// TIA Portal project "LF_project" (V16)

(* hardware
DEVICE "S7-1200 station_1"  S7-1200 Station
   slot 0: "Rack_0"  S7-1200 Rack  Rack  V1.0
   slot 1: "PLC_1"  CPU 1214C DC/DC/DC  6ES7 214-1AG40-0XB0  V4.2
   slot 2: "DI 16/DQ 16x24VDC_1"  6ES7 223-1BL32-0XB0  V2.0
   slot 3: "DI 16/DQ 16x24VDC_2"  6ES7 223-1BL32-0XB0  V2.0
   slot 4: "DI 16/DQ 16x24VDC_3"  6ES7 223-1BL32-0XB0  V2.0
   slot 5: "DI 16/DQ 16x24VDC_4"  6ES7 223-1BL32-0XB0  V2.0
   slot 6: "DI 16/DQ 16x24VDC_5"  6ES7 223-1BL32-0XB0  V2.0
   slot 7: "DI 16/DQ 16x24VDC_6"  6ES7 223-1BL32-0XB0  V2.0
*)

// ===== PLC "PLC_1"  CPU 1214C DC/DC/DC =====

VAR_GLOBAL   // PLC tag table "Default tag table"
   "System_Byte" AT %MB1 : Byte;
   "FirstScan" AT %M1.0 : Bool;
   "DiagStatusUpdate" AT %M1.1 : Bool;
   "AlwaysTRUE" AT %M1.2 : Bool;
   "AlwaysFALSE" AT %M1.3 : Bool;
END_VAR

VAR_GLOBAL   // PLC tag table "Input tags_1"
   "IN_1-0.0" AT %I0.0 : Bool;
   "IN_1-0.1" AT %I0.1 : Bool;
   "IN_1-0.2" AT %I0.2 : Bool;
   "IN_1-0.3" AT %I0.3 : Bool;
   "IN_1-0.4" AT %I0.4 : Bool;
   "IN_1-0.5" AT %I0.5 : Bool;
   "IN_1-0.6" AT %I0.6 : Bool;
   "IN_1-0.7" AT %I0.7 : Bool;
   "IN_1-1.0" AT %I1.0 : Bool;
   "IN_1-1.1" AT %I1.1 : Bool;
   "IN_1-1.2" AT %I1.2 : Bool;
   "IN_1-1.3" AT %I1.3 : Bool;
   "IN_1-1.4" AT %I1.4 : Bool;
   "IN_1-1.5" AT %I1.5 : Bool;
END_VAR

VAR_GLOBAL   // PLC tag table "Output tags_1"
   "OUT_1-0.0" AT %Q0.0 : Bool;
   "OUT_1-0.1" AT %Q0.1 : Bool;
   "OUT_1-0.2" AT %Q0.2 : Bool;
   "OUT_1-0.3" AT %Q0.3 : Bool;
   "OUT_1-0.4" AT %Q0.4 : Bool;
   "OUT_1-0.5" AT %Q0.5 : Bool;
   "OUT_1-0.6" AT %Q0.6 : Bool;
   "OUT_1-0.7" AT %Q0.7 : Bool;
   "OUT_1-1.0" AT %Q1.0 : Bool;
   "OUT_1-1.1" AT %Q1.1 : Bool;
END_VAR

VAR_GLOBAL   // PLC tag table "Input tags_2"
   "IN_2-0.0" AT %I8.0 : Bool;
   "IN_2-0.1" AT %I8.1 : Bool;
   "IN_2-0.2" AT %I8.2 : Bool;
   "IN_2-0.3" AT %I8.3 : Bool;
   "IN_2-0.4" AT %I8.4 : Bool;
   "IN_2-0.5" AT %I8.5 : Bool;
   "IN_2-0.6" AT %I8.6 : Bool;
   "IN_2-0.7" AT %I8.7 : Bool;
   "IN_2-1.0" AT %I9.0 : Bool;
   "IN_2-1.1" AT %I9.1 : Bool;
   "IN_2-1.2" AT %I9.2 : Bool;
   "IN_2-1.3" AT %I9.3 : Bool;
   "IN_2-1.4" AT %I9.4 : Bool;
   "IN_2-1.5" AT %I9.5 : Bool;
   "IN_2-1.6" AT %I9.6 : Bool;
   "IN_2-1.7" AT %I9.7 : Bool;
END_VAR

VAR_GLOBAL   // PLC tag table "Output tags_2"
   "OUT_2-0.0" AT %Q8.0 : Bool;
   "OUT_2-0.1" AT %Q8.1 : Bool;
   "OUT_2-0.2" AT %Q8.2 : Bool;
   "OUT_2-0.3" AT %Q8.3 : Bool;
   "OUT_2-0.4" AT %Q8.4 : Bool;
   "OUT_2-0.5" AT %Q8.5 : Bool;
   "OUT_2-0.6" AT %Q8.6 : Bool;
   "OUT_2-0.7" AT %Q8.7 : Bool;
   "OUT_2-1.0" AT %Q9.0 : Bool;
   "OUT_2-1.1" AT %Q9.1 : Bool;
   "OUT_2-1.2" AT %Q9.2 : Bool;
   "OUT_2-1.3" AT %Q9.3 : Bool;
   "OUT_2-1.4" AT %Q9.4 : Bool;
   "OUT_2-1.5" AT %Q9.5 : Bool;
   "OUT_2-1.6" AT %Q9.6 : Bool;
   "OUT_2-1.7" AT %Q9.7 : Bool;
END_VAR

VAR_GLOBAL   // PLC tag table "Input tags_3"
   "IN_3-0.0" AT %I12.0 : Bool;
   "IN_3-0.1" AT %I12.1 : Bool;
   "IN_3-0.2" AT %I12.2 : Bool;
   "IN_3-0.3" AT %I12.3 : Bool;
   "IN_3-0.4" AT %I12.4 : Bool;
   "IN_3-0.5" AT %I12.5 : Bool;
   "IN_3-0.6" AT %I12.6 : Bool;
   "IN_3-0.7" AT %I12.7 : Bool;
   "IN_3-1.0" AT %I13.0 : Bool;
   "IN_3-1.1" AT %I13.1 : Bool;
   "IN_3-1.2" AT %I13.2 : Bool;
   "IN_3-1.3" AT %I13.3 : Bool;
   "IN_3-1.4" AT %I13.4 : Bool;
   "IN_3-1.5" AT %I13.5 : Bool;
   "IN_3-1.6" AT %I13.6 : Bool;
   "IN_3-1.7" AT %I13.7 : Bool;
END_VAR

VAR_GLOBAL   // PLC tag table "Output tags_3"
   "OUT_3-0.0" AT %Q12.0 : Bool;
   "OUT_3-0.1" AT %Q12.1 : Bool;
   "OUT_3-0.2" AT %Q12.2 : Bool;
   "OUT_3-0.3" AT %Q12.3 : Bool;
   "OUT_3-0.4" AT %Q12.4 : Bool;
   "OUT_3-0.5" AT %Q12.5 : Bool;
   "OUT_3-0.6" AT %Q12.6 : Bool;
   "OUT_3-0.7" AT %Q12.7 : Bool;
   "OUT_3-1.0" AT %Q13.0 : Bool;
   "OUT_3-1.1" AT %Q13.1 : Bool;
   "OUT_3-1.2" AT %Q13.2 : Bool;
   "OUT_3-1.3" AT %Q13.3 : Bool;
   "OUT_3-1.4" AT %Q13.4 : Bool;
   "OUT_3-1.5" AT %Q13.5 : Bool;
   "OUT_3-1.6" AT %Q13.6 : Bool;
   "OUT_3-1.7" AT %Q13.7 : Bool;
END_VAR

VAR_GLOBAL   // PLC tag table "Input tags_4"
   "IN_4-0.0" AT %I16.0 : Bool;
   "IN_4-0.1" AT %I16.1 : Bool;
   "IN_4-0.2" AT %I16.2 : Bool;
   "IN_4-0.3" AT %I16.3 : Bool;
   "IN_4-0.4" AT %I16.4 : Bool;
   "IN_4-0.5" AT %I16.5 : Bool;
   "IN_4-0.6" AT %I16.6 : Bool;
   "IN_4-0.7" AT %I16.7 : Bool;
   "IN_4-1.0" AT %I17.0 : Bool;
   "IN_4-1.1" AT %I17.1 : Bool;
   "IN_4-1.2" AT %I17.2 : Bool;
   "IN_4-1.3" AT %I17.3 : Bool;
   "IN_4-1.4" AT %I17.4 : Bool;
   "IN_4-1.5" AT %I17.5 : Bool;
   "IN_4-1.6" AT %I17.6 : Bool;
   "IN_4-1.7" AT %I17.7 : Bool;
END_VAR

VAR_GLOBAL   // PLC tag table "Output tags_4"
   "OUT_4-0.0" AT %Q16.0 : Bool;
   "OUT_4-0.1" AT %Q16.1 : Bool;
   "OUT_4-0.2" AT %Q16.2 : Bool;
   "OUT_4-0.3" AT %Q16.3 : Bool;
   "OUT_4-0.4" AT %Q16.4 : Bool;
   "OUT_4-0.5" AT %Q16.5 : Bool;
   "OUT_4-0.6" AT %Q16.6 : Bool;
   "OUT_4-0.7" AT %Q16.7 : Bool;
   "OUT_4-1.0" AT %Q17.0 : Bool;
   "OUT_4-1.1" AT %Q17.1 : Bool;
   "OUT_4-1.2" AT %Q17.2 : Bool;
   "OUT_4-1.3" AT %Q17.3 : Bool;
   "OUT_4-1.4" AT %Q17.4 : Bool;
   "OUT_4-1.5" AT %Q17.5 : Bool;
   "OUT_4-1.6" AT %Q17.6 : Bool;
   "OUT_4-1.7" AT %Q17.7 : Bool;
END_VAR

VAR_GLOBAL   // PLC tag table "Input tags_5"
   "IN_5-0.0" AT %I20.0 : Bool;
   "IN_5-0.1" AT %I20.1 : Bool;
   "IN_5-0.2" AT %I20.2 : Bool;
   "IN_5-0.3" AT %I20.3 : Bool;
   "IN_5-0.4" AT %I20.4 : Bool;
   "IN_5-0.5" AT %I20.5 : Bool;
   "IN_5-0.6" AT %I20.6 : Bool;
   "IN_5-0.7" AT %I20.7 : Bool;
   "IN_5-1.0" AT %I21.0 : Bool;
   "IN_5-1.1" AT %I21.1 : Bool;
   "IN_5-1.2" AT %I21.2 : Bool;
   "IN_5-1.3" AT %I21.3 : Bool;
   "IN_5-1.4" AT %I21.4 : Bool;
   "IN_5-1.5" AT %I21.5 : Bool;
   "IN_5-1.6" AT %I21.6 : Bool;
   "IN_5-1.7" AT %I21.7 : Bool;
END_VAR

VAR_GLOBAL   // PLC tag table "Output tags_5"
   "OUT_5-0.0" AT %Q20.0 : Bool;
   "OUT_5-0.1" AT %Q20.1 : Bool;
   "OUT_5-0.2" AT %Q20.2 : Bool;
   "OUT_5-0.3" AT %Q20.3 : Bool;
   "OUT_5-0.4" AT %Q20.4 : Bool;
   "OUT_5-0.5" AT %Q20.5 : Bool;
   "OUT_5-0.6" AT %Q20.6 : Bool;
   "OUT_5-0.7" AT %Q20.7 : Bool;
   "OUT_5-1.0" AT %Q21.0 : Bool;
   "OUT_5-1.1" AT %Q21.1 : Bool;
   "OUT_5-1.2" AT %Q21.2 : Bool;
   "OUT_5-1.3" AT %Q21.3 : Bool;
   "OUT_5-1.4" AT %Q21.4 : Bool;
   "OUT_5-1.5" AT %Q21.5 : Bool;
   "OUT_5-1.6" AT %Q21.6 : Bool;
   "OUT_5-1.7" AT %Q21.7 : Bool;
END_VAR

VAR_GLOBAL   // PLC tag table "Input tags_6"
   "IN_6-0.0" AT %I24.0 : Bool;
   "IN_6-0.1" AT %I24.1 : Bool;
   "IN_6-0.2" AT %I24.2 : Bool;
   "IN_6-0.3" AT %I24.3 : Bool;
   "IN_6-0.4" AT %I24.4 : Bool;
   "IN_6-0.5" AT %I24.5 : Bool;
   "IN_6-0.6" AT %I24.6 : Bool;
   "IN_6-0.7" AT %I24.7 : Bool;
   "IN_6-1.0" AT %I25.0 : Bool;
   "IN_6-1.1" AT %I25.1 : Bool;
   "IN_6-1.2" AT %I25.2 : Bool;
   "IN_6-1.3" AT %I25.3 : Bool;
   "IN_6-1.4" AT %I25.4 : Bool;
   "IN_6-1.5" AT %I25.5 : Bool;
   "IN_6-1.6" AT %I25.6 : Bool;
   "IN_6-1.7" AT %I25.7 : Bool;
END_VAR

VAR_GLOBAL   // PLC tag table "Output tags_6"
   "OUT_6-0.0" AT %Q24.0 : Bool;
   "OUT_6-0.1" AT %Q24.1 : Bool;
   "OUT_6-0.2" AT %Q24.2 : Bool;
   "OUT_6-0.3" AT %Q24.3 : Bool;
   "OUT_6-0.4" AT %Q24.4 : Bool;
   "OUT_6-0.5" AT %Q24.5 : Bool;
   "OUT_6-0.6" AT %Q24.6 : Bool;
   "OUT_6-0.7" AT %Q24.7 : Bool;
   "OUT_6-1.0" AT %Q25.0 : Bool;
   "OUT_6-1.1" AT %Q25.1 : Bool;
   "OUT_6-1.2" AT %Q25.2 : Bool;
   "OUT_6-1.3" AT %Q25.3 : Bool;
   "OUT_6-1.4" AT %Q25.4 : Bool;
   "OUT_6-1.5" AT %Q25.5 : Bool;
   "OUT_6-1.6" AT %Q25.6 : Bool;
   "OUT_6-1.7" AT %Q25.7 : Bool;
END_VAR

VAR_GLOBAL   // PLC tag table "Input tags_7"
   "IN_7-0.0" AT %I28.0 : Bool;
   "IN_7-0.1" AT %I28.1 : Bool;
   "IN_7-0.2" AT %I28.2 : Bool;
   "IN_7-0.3" AT %I28.3 : Bool;
   "IN_7-0.4" AT %I28.4 : Bool;
   "IN_7-0.5" AT %I28.5 : Bool;
   "IN_7-0.6" AT %I28.6 : Bool;
   "IN_7-0.7" AT %I28.7 : Bool;
   "IN_7-1.0" AT %I29.0 : Bool;
   "IN_7-1.1" AT %I29.1 : Bool;
   "IN_7-1.2" AT %I29.2 : Bool;
   "IN_7-1.3" AT %I29.3 : Bool;
   "IN_7-1.4" AT %I29.4 : Bool;
   "IN_7-1.5" AT %I29.5 : Bool;
   "IN_7-1.6" AT %I29.6 : Bool;
   "IN_7-1.7" AT %I29.7 : Bool;
END_VAR

VAR_GLOBAL   // PLC tag table "Output tags_7"
   "OUT_7-0.0" AT %Q28.0 : Bool;
   "OUT_7-0.1" AT %Q28.1 : Bool;
   "OUT_7-0.2" AT %Q28.2 : Bool;
   "OUT_7-0.3" AT %Q28.3 : Bool;
   "OUT_7-0.4" AT %Q28.4 : Bool;
   "OUT_7-0.5" AT %Q28.5 : Bool;
   "OUT_7-0.6" AT %Q28.6 : Bool;
   "OUT_7-0.7" AT %Q28.7 : Bool;
   "OUT_7-1.0" AT %Q29.0 : Bool;
   "OUT_7-1.1" AT %Q29.1 : Bool;
   "OUT_7-1.2" AT %Q29.2 : Bool;
   "OUT_7-1.3" AT %Q29.3 : Bool;
   "OUT_7-1.4" AT %Q29.4 : Bool;
   "OUT_7-1.5" AT %Q29.5 : Bool;
   "OUT_7-1.6" AT %Q29.6 : Bool;
   "OUT_7-1.7" AT %Q29.7 : Bool;
END_VAR

VAR_GLOBAL   // PLC tag table "Analog tags"
   "AN_1" AT %IW64 : Int;
   "AN_2" AT %IW66 : Int;
END_VAR

DATA_BLOCK "MODBUS"   // DB1
{ S7_Optimized_Access := 'FALSE' }
VERSION : 0.1
   VAR
      PLC_ports : Struct
         Analogs : Array[0..1] of Word;
         Inputs : Array[0..109] of Word;
         Outputs : Array[0..105] of Word;
      END_STRUCT;
      Connection : TCON_IP_v4;
   END_VAR
BEGIN
   Connection.InterfaceId := 64;
   Connection.ID := 1;
   Connection.ConnectionType := 11;
   Connection.LocalPort := 502;
END_DATA_BLOCK

DATA_BLOCK "Algorythm_DB"   // DB6
{ S7_Optimized_Access := 'TRUE' }
VERSION : 0.1
// stored: InstanceOfName Algorythm
"Algorythm"
BEGIN
END_DATA_BLOCK

// folder: Loaders

DATA_BLOCK "Loader 0_DB"   // DB7
{ S7_Optimized_Access := 'TRUE' }
VERSION : 0.1
// stored: InstanceOfName Loader 0
"Loader 0"
BEGIN
END_DATA_BLOCK

DATA_BLOCK "Loader 1_DB"   // DB8
{ S7_Optimized_Access := 'TRUE' }
VERSION : 0.1
// stored: InstanceOfName Loader 1
"Loader 1"
BEGIN
END_DATA_BLOCK

// folder: PLC signals

DATA_BLOCK "Analog signals_DB"   // DB3
{ S7_Optimized_Access := 'TRUE' }
VERSION : 0.1
// stored: InstanceOfName Analog signals
"Analog signals"
BEGIN
END_DATA_BLOCK

DATA_BLOCK "Input signals_DB"   // DB4
{ S7_Optimized_Access := 'TRUE' }
VERSION : 0.1
// stored: InstanceOfName Input signals
"Input signals"
BEGIN
END_DATA_BLOCK

DATA_BLOCK "Output signals_DB"   // DB5
{ S7_Optimized_Access := 'TRUE' }
VERSION : 0.1
// stored: InstanceOfName Output signals
"Output signals"
BEGIN
END_DATA_BLOCK

// folder: System blocks/Program resources

DATA_BLOCK "IEC_Timer_0_DB"   // DB20
{ S7_Optimized_Access := 'TRUE' }
AUTHOR : Simatic
FAMILY : IEC
NAME : IEC_TMR
VERSION : 1.0
// stored: InstanceOfName IEC_TIMER
"IEC_TIMER"
BEGIN
END_DATA_BLOCK

// folder: (top level)

FUNCTION_BLOCK "Algorythm"   // FB4, LAD
{ S7_Optimized_Access := 'TRUE' }
VERSION : 0.1
   VAR
      var : Array[0..100] of Bool;
   END_VAR
   VAR_TEMP
      i : Bool;
   END_VAR
   VAR_TEMP   // added for the SCL form of the ladder/FBD networks
      _w1 : Bool;
      _w2 : Bool;
      _w3 : Bool;
      _w4 : Bool;
      _w5 : Bool;
      _w6 : Bool;
      _w7 : Bool;
      _w8 : Bool;
      _w9 : Bool;
   END_VAR
BEGIN

REGION Network 1
   // Функция - доставка груза грузчиком 0:
   // var[0] - OUT_1-0.3, подъехать
   // var[1] - OUT_1-0.5, подняться
   // var[2] - OUT_1-1.0, выдвинуться
   // var[3] - OUT_1-0.5, приподняться
   // var[4] - OUT_1-0.7, задвинуться
   // var[5] - OUT_1-0.2, подъехать
   // var[6] - OUT_1-0.7, выдвинуться
   // var[7] - OUT_1-0.6, опуститься
   // .......................................................
   // var[10] - OUT_1-0.5, подняться
   // var[11] - OUT_1-1.0, задвинуться
   // 
   // Поясняющие диапазоны:
   // (1-0.2 - 1-1.5) - туда-сюда
   // (2-0.1 - 2-1.0) - вверх-вниз
   // (2-1.1 - 2-1.3) - влево-вправо
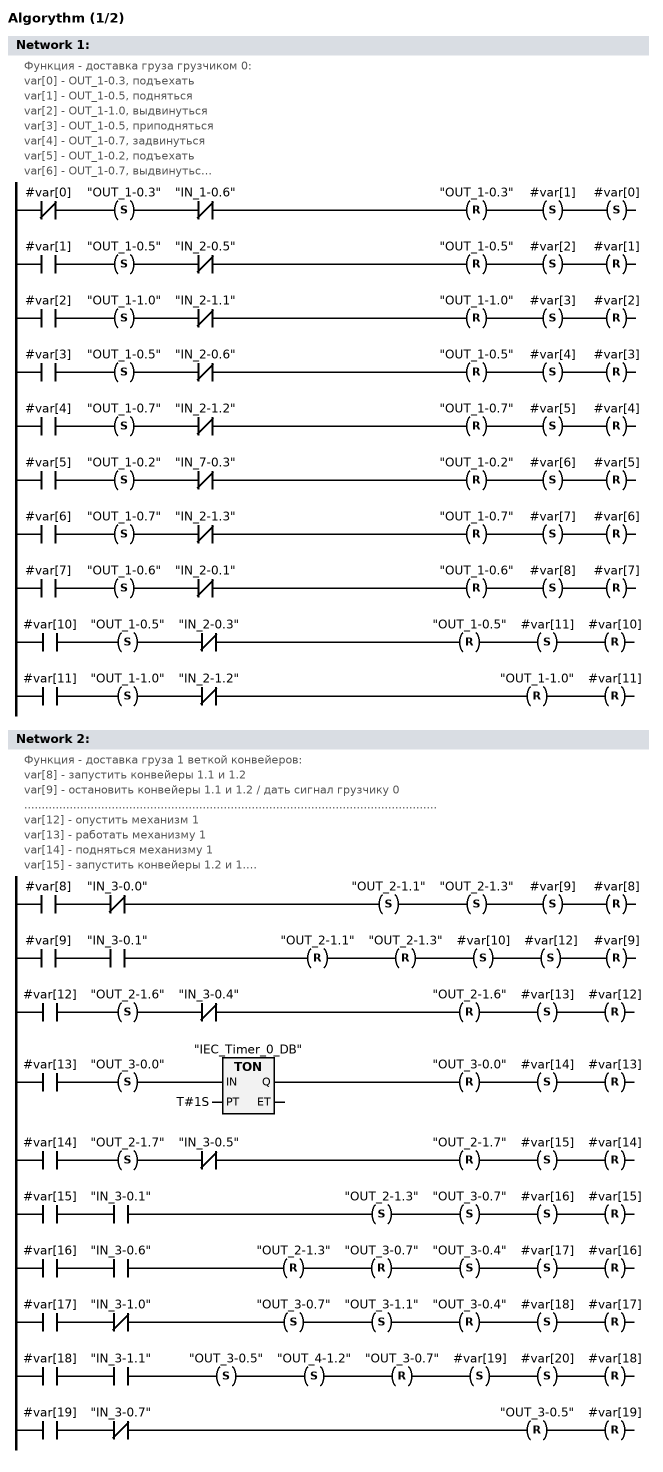
   RUNG wire#powerrail
      I_Contact( #var[0] )
      S_Coil( "OUT_1-0.3" )
      I_Contact( "IN_1-0.6" )
      R_Coil( "OUT_1-0.3" )
      S_Coil( #var[1] )
      S_Coil( #var[0] )
   END_RUNG
   RUNG wire#powerrail
      Contact( #var[1] )
      S_Coil( "OUT_1-0.5" )
      I_Contact( "IN_2-0.5" )
      R_Coil( "OUT_1-0.5" )
      S_Coil( #var[2] )
      R_Coil( #var[1] )
   END_RUNG
   RUNG wire#powerrail
      Contact( #var[2] )
      S_Coil( "OUT_1-1.0" )
      I_Contact( "IN_2-1.1" )
      R_Coil( "OUT_1-1.0" )
      S_Coil( #var[3] )
      R_Coil( #var[2] )
   END_RUNG
   RUNG wire#powerrail
      Contact( #var[3] )
      S_Coil( "OUT_1-0.5" )
      I_Contact( "IN_2-0.6" )
      R_Coil( "OUT_1-0.5" )
      S_Coil( #var[4] )
      R_Coil( #var[3] )
   END_RUNG
   RUNG wire#powerrail
      Contact( #var[4] )
      S_Coil( "OUT_1-0.7" )
      I_Contact( "IN_2-1.2" )
      R_Coil( "OUT_1-0.7" )
      S_Coil( #var[5] )
      R_Coil( #var[4] )
   END_RUNG
   RUNG wire#powerrail
      Contact( #var[5] )
      S_Coil( "OUT_1-0.2" )
      I_Contact( "IN_7-0.3" )
      R_Coil( "OUT_1-0.2" )
      S_Coil( #var[6] )
      R_Coil( #var[5] )
   END_RUNG
   RUNG wire#powerrail
      Contact( #var[6] )
      S_Coil( "OUT_1-0.7" )
      I_Contact( "IN_2-1.3" )
      R_Coil( "OUT_1-0.7" )
      S_Coil( #var[7] )
      R_Coil( #var[6] )
   END_RUNG
   RUNG wire#powerrail
      Contact( #var[7] )
      S_Coil( "OUT_1-0.6" )
      I_Contact( "IN_2-0.1" )
      R_Coil( "OUT_1-0.6" )
      S_Coil( #var[8] )
      R_Coil( #var[7] )
   END_RUNG
   RUNG wire#powerrail
      Contact( #var[10] )
      S_Coil( "OUT_1-0.5" )
      I_Contact( "IN_2-0.3" )
      R_Coil( "OUT_1-0.5" )
      S_Coil( #var[11] )
      R_Coil( #var[10] )
   END_RUNG
   RUNG wire#powerrail
      Contact( #var[11] )
      S_Coil( "OUT_1-1.0" )
      I_Contact( "IN_2-1.2" )
      R_Coil( "OUT_1-1.0" )
      R_Coil( #var[11] )
   END_RUNG
   // the same network as SCL:
   IF NOT #var[0] THEN "OUT_1-0.3" := TRUE; END_IF;
   IF NOT #var[0] AND NOT "IN_1-0.6" THEN "OUT_1-0.3" := FALSE; END_IF;
   #_w1 := NOT #var[0] AND NOT "IN_1-0.6";
   IF #_w1 THEN
       #var[1] := TRUE;
       #var[0] := TRUE;
   END_IF;
   IF #var[1] THEN "OUT_1-0.5" := TRUE; END_IF;
   IF #var[1] AND NOT "IN_2-0.5" THEN "OUT_1-0.5" := FALSE; END_IF;
   #_w2 := #var[1] AND NOT "IN_2-0.5";
   IF #_w2 THEN
       #var[2] := TRUE;
       #var[1] := FALSE;
   END_IF;
   IF #var[2] THEN "OUT_1-1.0" := TRUE; END_IF;
   IF #var[2] AND NOT "IN_2-1.1" THEN "OUT_1-1.0" := FALSE; END_IF;
   #_w3 := #var[2] AND NOT "IN_2-1.1";
   IF #_w3 THEN
       #var[3] := TRUE;
       #var[2] := FALSE;
   END_IF;
   IF #var[3] THEN "OUT_1-0.5" := TRUE; END_IF;
   IF #var[3] AND NOT "IN_2-0.6" THEN "OUT_1-0.5" := FALSE; END_IF;
   #_w4 := #var[3] AND NOT "IN_2-0.6";
   IF #_w4 THEN
       #var[4] := TRUE;
       #var[3] := FALSE;
   END_IF;
   IF #var[4] THEN "OUT_1-0.7" := TRUE; END_IF;
   IF #var[4] AND NOT "IN_2-1.2" THEN "OUT_1-0.7" := FALSE; END_IF;
   #_w5 := #var[4] AND NOT "IN_2-1.2";
   IF #_w5 THEN
       #var[5] := TRUE;
       #var[4] := FALSE;
   END_IF;
   IF #var[5] THEN "OUT_1-0.2" := TRUE; END_IF;
   IF #var[5] AND NOT "IN_7-0.3" THEN "OUT_1-0.2" := FALSE; END_IF;
   #_w6 := #var[5] AND NOT "IN_7-0.3";
   IF #_w6 THEN
       #var[6] := TRUE;
       #var[5] := FALSE;
   END_IF;
   IF #var[6] THEN "OUT_1-0.7" := TRUE; END_IF;
   IF #var[6] AND NOT "IN_2-1.3" THEN "OUT_1-0.7" := FALSE; END_IF;
   #_w7 := #var[6] AND NOT "IN_2-1.3";
   IF #_w7 THEN
       #var[7] := TRUE;
       #var[6] := FALSE;
   END_IF;
   IF #var[7] THEN "OUT_1-0.6" := TRUE; END_IF;
   IF #var[7] AND NOT "IN_2-0.1" THEN "OUT_1-0.6" := FALSE; END_IF;
   #_w8 := #var[7] AND NOT "IN_2-0.1";
   IF #_w8 THEN
       #var[8] := TRUE;
       #var[7] := FALSE;
   END_IF;
   IF #var[10] THEN "OUT_1-0.5" := TRUE; END_IF;
   IF #var[10] AND NOT "IN_2-0.3" THEN "OUT_1-0.5" := FALSE; END_IF;
   #_w9 := #var[10] AND NOT "IN_2-0.3";
   IF #_w9 THEN
       #var[11] := TRUE;
       #var[10] := FALSE;
   END_IF;
   IF #var[11] THEN "OUT_1-1.0" := TRUE; END_IF;
   IF #var[11] AND NOT "IN_2-1.2" THEN
       "OUT_1-1.0" := FALSE;
       #var[11] := FALSE;
   END_IF;
END_REGION

REGION Network 2
   // Функция - доставка груза 1 веткой конвейеров:
   // var[8] - запустить конвейеры 1.1 и 1.2
   // var[9] - остановить конвейеры 1.1 и 1.2 / дать сигнал грузчику 0
   // ......................................................................................................................
   // var[12] - опустить механизм 1
   // var[13] - работать механизму 1
   // var[14] - подняться механизму 1
   // var[15] - запустить конвейеры 1.2 и 1.3
   // var[16] - остановить конвейеры 1.2 и 1.3 / запустить поворот конвейера 1.3
   // var[17] - запустить конвейеры 1.3 и 1.4 / остановить поворот конвейера 1.3
   // var[18] - остановить конвейер 1.3 / запустить конвейер 2.3 / запустить поворот конвейера 1.3
   // var[19] - остановить поворот конвейера 1.3
   IF #var[8] AND NOT "IN_3-0.0" THEN
       "OUT_2-1.1" := TRUE;
       "OUT_2-1.3" := TRUE;
   END_IF;
   #_w1 := #var[8] AND NOT "IN_3-0.0";
   IF #_w1 THEN
       #var[9] := TRUE;
       #var[8] := FALSE;
   END_IF;
   IF #var[9] AND "IN_3-0.1" THEN
       "OUT_2-1.1" := FALSE;
       "OUT_2-1.3" := FALSE;
   END_IF;
   #_w2 := #var[9] AND "IN_3-0.1";
   IF #_w2 THEN
       #var[10] := TRUE;
       #var[12] := TRUE;
       #var[9] := FALSE;
   END_IF;
   IF #var[12] THEN "OUT_2-1.6" := TRUE; END_IF;
   IF #var[12] AND NOT "IN_3-0.4" THEN "OUT_2-1.6" := FALSE; END_IF;
   #_w3 := #var[12] AND NOT "IN_3-0.4";
   IF #_w3 THEN
       #var[13] := TRUE;
       #var[12] := FALSE;
   END_IF;
   IF #var[13] THEN "OUT_3-0.0" := TRUE; END_IF;
   "IEC_Timer_0_DB".TON(IN := #var[13], PT := T#1S);
   IF "IEC_Timer_0_DB".Q THEN
       "OUT_3-0.0" := FALSE;
       #var[14] := TRUE;
       #var[13] := FALSE;
   END_IF;
   IF #var[14] THEN "OUT_2-1.7" := TRUE; END_IF;
   IF #var[14] AND NOT "IN_3-0.5" THEN "OUT_2-1.7" := FALSE; END_IF;
   #_w4 := #var[14] AND NOT "IN_3-0.5";
   IF #_w4 THEN
       #var[15] := TRUE;
       #var[14] := FALSE;
   END_IF;
   IF #var[15] AND "IN_3-0.1" THEN
       "OUT_2-1.3" := TRUE;
       "OUT_3-0.7" := TRUE;
   END_IF;
   #_w5 := #var[15] AND "IN_3-0.1";
   IF #_w5 THEN
       #var[16] := TRUE;
       #var[15] := FALSE;
   END_IF;
   IF #var[16] AND "IN_3-0.6" THEN
       "OUT_2-1.3" := FALSE;
       "OUT_3-0.7" := FALSE;
       "OUT_3-0.4" := TRUE;
   END_IF;
   #_w6 := #var[16] AND "IN_3-0.6";
   IF #_w6 THEN
       #var[17] := TRUE;
       #var[16] := FALSE;
   END_IF;
   IF #var[17] AND NOT "IN_3-1.0" THEN
       "OUT_3-0.7" := TRUE;
       "OUT_3-1.1" := TRUE;
       "OUT_3-0.4" := FALSE;
   END_IF;
   #_w7 := #var[17] AND NOT "IN_3-1.0";
   IF #_w7 THEN
       #var[18] := TRUE;
       #var[17] := FALSE;
   END_IF;
   IF #var[18] AND "IN_3-1.1" THEN
       "OUT_3-0.5" := TRUE;
       "OUT_4-1.2" := TRUE;
       "OUT_3-0.7" := FALSE;
   END_IF;
   #_w8 := #var[18] AND "IN_3-1.1";
   IF #_w8 THEN
       #var[19] := TRUE;
       #var[20] := TRUE;
       #var[18] := FALSE;
   END_IF;
   IF #var[19] AND NOT "IN_3-0.7" THEN
       "OUT_3-0.5" := FALSE;
       #var[19] := FALSE;
   END_IF;
END_REGION

REGION Network 3
   // Функция - доставка груза 2 веткой конвейеров:
   // var[20] - остановить конвейер 1.4 / запустить конвейер 2.4
   // var[21] - остановить конвейер 2.3 / запустить конвейер 3.3
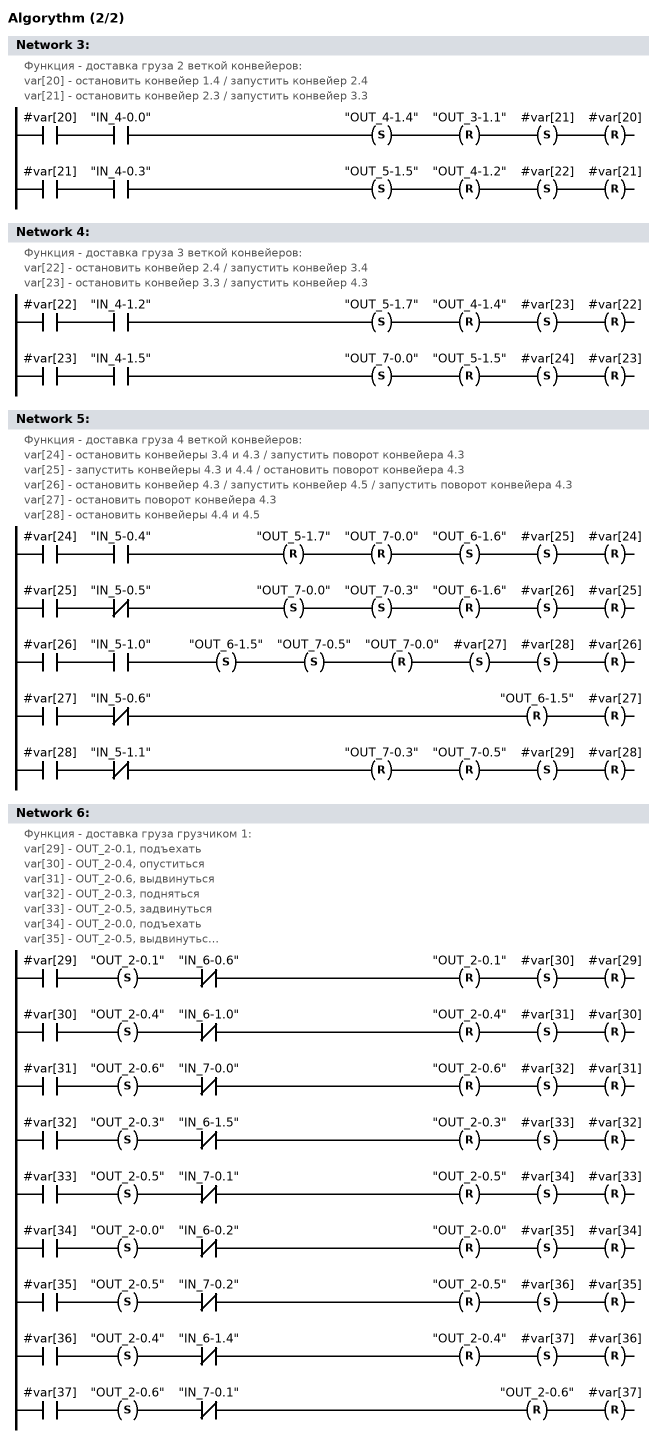
   RUNG wire#powerrail
      Contact( #var[20] )
      Contact( "IN_4-0.0" )
      S_Coil( "OUT_4-1.4" )
      R_Coil( "OUT_3-1.1" )
      S_Coil( #var[21] )
      R_Coil( #var[20] )
   END_RUNG
   RUNG wire#powerrail
      Contact( #var[21] )
      Contact( "IN_4-0.3" )
      S_Coil( "OUT_5-1.5" )
      R_Coil( "OUT_4-1.2" )
      S_Coil( #var[22] )
      R_Coil( #var[21] )
   END_RUNG
   // the same network as SCL:
   IF #var[20] AND "IN_4-0.0" THEN
       "OUT_4-1.4" := TRUE;
       "OUT_3-1.1" := FALSE;
   END_IF;
   #_w1 := #var[20] AND "IN_4-0.0";
   IF #_w1 THEN
       #var[21] := TRUE;
       #var[20] := FALSE;
   END_IF;
   IF #var[21] AND "IN_4-0.3" THEN
       "OUT_5-1.5" := TRUE;
       "OUT_4-1.2" := FALSE;
   END_IF;
   #_w2 := #var[21] AND "IN_4-0.3";
   IF #_w2 THEN
       #var[22] := TRUE;
       #var[21] := FALSE;
   END_IF;
END_REGION

REGION Network 4
   // Функция - доставка груза 3 веткой конвейеров:
   // var[22] - остановить конвейер 2.4 / запустить конвейер 3.4
   // var[23] - остановить конвейер 3.3 / запустить конвейер 4.3
   RUNG wire#powerrail
      Contact( #var[22] )
      Contact( "IN_4-1.2" )
      S_Coil( "OUT_5-1.7" )
      R_Coil( "OUT_4-1.4" )
      S_Coil( #var[23] )
      R_Coil( #var[22] )
   END_RUNG
   RUNG wire#powerrail
      Contact( #var[23] )
      Contact( "IN_4-1.5" )
      S_Coil( "OUT_7-0.0" )
      R_Coil( "OUT_5-1.5" )
      S_Coil( #var[24] )
      R_Coil( #var[23] )
   END_RUNG
   // the same network as SCL:
   IF #var[22] AND "IN_4-1.2" THEN
       "OUT_5-1.7" := TRUE;
       "OUT_4-1.4" := FALSE;
   END_IF;
   #_w1 := #var[22] AND "IN_4-1.2";
   IF #_w1 THEN
       #var[23] := TRUE;
       #var[22] := FALSE;
   END_IF;
   IF #var[23] AND "IN_4-1.5" THEN
       "OUT_7-0.0" := TRUE;
       "OUT_5-1.5" := FALSE;
   END_IF;
   #_w2 := #var[23] AND "IN_4-1.5";
   IF #_w2 THEN
       #var[24] := TRUE;
       #var[23] := FALSE;
   END_IF;
END_REGION

REGION Network 5
   // Функция - доставка груза 4 веткой конвейеров:
   // var[24] - остановить конвейеры 3.4 и 4.3 / запустить поворот конвейера 4.3
   // var[25] - запустить конвейеры 4.3 и 4.4 / остановить поворот конвейера 4.3
   // var[26] - остановить конвейер 4.3 / запустить конвейер 4.5 / запустить поворот конвейера 4.3
   // var[27] - остановить поворот конвейера 4.3
   // var[28] - остановить конвейеры 4.4 и 4.5
   RUNG wire#powerrail
      Contact( #var[24] )
      Contact( "IN_5-0.4" )
      R_Coil( "OUT_5-1.7" )
      R_Coil( "OUT_7-0.0" )
      S_Coil( "OUT_6-1.6" )
      S_Coil( #var[25] )
      R_Coil( #var[24] )
   END_RUNG
   RUNG wire#powerrail
      Contact( #var[25] )
      I_Contact( "IN_5-0.5" )
      S_Coil( "OUT_7-0.0" )
      S_Coil( "OUT_7-0.3" )
      R_Coil( "OUT_6-1.6" )
      S_Coil( #var[26] )
      R_Coil( #var[25] )
   END_RUNG
   RUNG wire#powerrail
      Contact( #var[26] )
      Contact( "IN_5-1.0" )
      S_Coil( "OUT_6-1.5" )
      S_Coil( "OUT_7-0.5" )
      R_Coil( "OUT_7-0.0" )
      S_Coil( #var[27] )
      S_Coil( #var[28] )
      R_Coil( #var[26] )
   END_RUNG
   RUNG wire#powerrail
      Contact( #var[27] )
      I_Contact( "IN_5-0.6" )
      R_Coil( "OUT_6-1.5" )
      R_Coil( #var[27] )
   END_RUNG
   RUNG wire#powerrail
      Contact( #var[28] )
      I_Contact( "IN_5-1.1" )
      R_Coil( "OUT_7-0.3" )
      R_Coil( "OUT_7-0.5" )
      S_Coil( #var[29] )
      R_Coil( #var[28] )
   END_RUNG
   // the same network as SCL:
   IF #var[24] AND "IN_5-0.4" THEN
       "OUT_5-1.7" := FALSE;
       "OUT_7-0.0" := FALSE;
       "OUT_6-1.6" := TRUE;
   END_IF;
   #_w1 := #var[24] AND "IN_5-0.4";
   IF #_w1 THEN
       #var[25] := TRUE;
       #var[24] := FALSE;
   END_IF;
   IF #var[25] AND NOT "IN_5-0.5" THEN
       "OUT_7-0.0" := TRUE;
       "OUT_7-0.3" := TRUE;
       "OUT_6-1.6" := FALSE;
   END_IF;
   #_w2 := #var[25] AND NOT "IN_5-0.5";
   IF #_w2 THEN
       #var[26] := TRUE;
       #var[25] := FALSE;
   END_IF;
   IF #var[26] AND "IN_5-1.0" THEN
       "OUT_6-1.5" := TRUE;
       "OUT_7-0.5" := TRUE;
       "OUT_7-0.0" := FALSE;
   END_IF;
   #_w3 := #var[26] AND "IN_5-1.0";
   IF #_w3 THEN
       #var[27] := TRUE;
       #var[28] := TRUE;
       #var[26] := FALSE;
   END_IF;
   IF #var[27] AND NOT "IN_5-0.6" THEN
       "OUT_6-1.5" := FALSE;
       #var[27] := FALSE;
   END_IF;
   IF #var[28] AND NOT "IN_5-1.1" THEN
       "OUT_7-0.3" := FALSE;
       "OUT_7-0.5" := FALSE;
   END_IF;
   #_w4 := #var[28] AND NOT "IN_5-1.1";
   IF #_w4 THEN
       #var[29] := TRUE;
       #var[28] := FALSE;
   END_IF;
END_REGION

REGION Network 6
   // Функция - доставка груза грузчиком 1:
   // var[29] - OUT_2-0.1, подъехать
   // var[30] - OUT_2-0.4, опуститься
   // var[31] - OUT_2-0.6, выдвинуться
   // var[32] - OUT_2-0.3, подняться
   // var[33] - OUT_2-0.5, задвинуться
   // var[34] - OUT_2-0.0, подъехать
   // var[35] - OUT_2-0.5, выдвинуться
   // var[36] - OUT_2-0.4, приспуститься
   // var[37] - OUT_2-0.6, задвинуться
   // 
   // Поясняющие диапазоны:
   // (5-1.3 - 6-0.6) - туда-сюда
   // (6-1.0 - 6-1.7) - вверх-вниз
   // (7-0.0 - 7-0.2) - влево-вправо
   RUNG wire#powerrail
      Contact( #var[29] )
      S_Coil( "OUT_2-0.1" )
      I_Contact( "IN_6-0.6" )
      R_Coil( "OUT_2-0.1" )
      S_Coil( #var[30] )
      R_Coil( #var[29] )
   END_RUNG
   RUNG wire#powerrail
      Contact( #var[30] )
      S_Coil( "OUT_2-0.4" )
      I_Contact( "IN_6-1.0" )
      R_Coil( "OUT_2-0.4" )
      S_Coil( #var[31] )
      R_Coil( #var[30] )
   END_RUNG
   RUNG wire#powerrail
      Contact( #var[31] )
      S_Coil( "OUT_2-0.6" )
      I_Contact( "IN_7-0.0" )
      R_Coil( "OUT_2-0.6" )
      S_Coil( #var[32] )
      R_Coil( #var[31] )
   END_RUNG
   RUNG wire#powerrail
      Contact( #var[32] )
      S_Coil( "OUT_2-0.3" )
      I_Contact( "IN_6-1.5" )
      R_Coil( "OUT_2-0.3" )
      S_Coil( #var[33] )
      R_Coil( #var[32] )
   END_RUNG
   RUNG wire#powerrail
      Contact( #var[33] )
      S_Coil( "OUT_2-0.5" )
      I_Contact( "IN_7-0.1" )
      R_Coil( "OUT_2-0.5" )
      S_Coil( #var[34] )
      R_Coil( #var[33] )
   END_RUNG
   RUNG wire#powerrail
      Contact( #var[34] )
      S_Coil( "OUT_2-0.0" )
      I_Contact( "IN_6-0.2" )
      R_Coil( "OUT_2-0.0" )
      S_Coil( #var[35] )
      R_Coil( #var[34] )
   END_RUNG
   RUNG wire#powerrail
      Contact( #var[35] )
      S_Coil( "OUT_2-0.5" )
      I_Contact( "IN_7-0.2" )
      R_Coil( "OUT_2-0.5" )
      S_Coil( #var[36] )
      R_Coil( #var[35] )
   END_RUNG
   RUNG wire#powerrail
      Contact( #var[36] )
      S_Coil( "OUT_2-0.4" )
      I_Contact( "IN_6-1.4" )
      R_Coil( "OUT_2-0.4" )
      S_Coil( #var[37] )
      R_Coil( #var[36] )
   END_RUNG
   RUNG wire#powerrail
      Contact( #var[37] )
      S_Coil( "OUT_2-0.6" )
      I_Contact( "IN_7-0.1" )
      R_Coil( "OUT_2-0.6" )
      R_Coil( #var[37] )
   END_RUNG
   // the same network as SCL:
   IF #var[29] THEN "OUT_2-0.1" := TRUE; END_IF;
   IF #var[29] AND NOT "IN_6-0.6" THEN "OUT_2-0.1" := FALSE; END_IF;
   #_w1 := #var[29] AND NOT "IN_6-0.6";
   IF #_w1 THEN
       #var[30] := TRUE;
       #var[29] := FALSE;
   END_IF;
   IF #var[30] THEN "OUT_2-0.4" := TRUE; END_IF;
   IF #var[30] AND NOT "IN_6-1.0" THEN "OUT_2-0.4" := FALSE; END_IF;
   #_w2 := #var[30] AND NOT "IN_6-1.0";
   IF #_w2 THEN
       #var[31] := TRUE;
       #var[30] := FALSE;
   END_IF;
   IF #var[31] THEN "OUT_2-0.6" := TRUE; END_IF;
   IF #var[31] AND NOT "IN_7-0.0" THEN "OUT_2-0.6" := FALSE; END_IF;
   #_w3 := #var[31] AND NOT "IN_7-0.0";
   IF #_w3 THEN
       #var[32] := TRUE;
       #var[31] := FALSE;
   END_IF;
   IF #var[32] THEN "OUT_2-0.3" := TRUE; END_IF;
   IF #var[32] AND NOT "IN_6-1.5" THEN "OUT_2-0.3" := FALSE; END_IF;
   #_w4 := #var[32] AND NOT "IN_6-1.5";
   IF #_w4 THEN
       #var[33] := TRUE;
       #var[32] := FALSE;
   END_IF;
   IF #var[33] THEN "OUT_2-0.5" := TRUE; END_IF;
   IF #var[33] AND NOT "IN_7-0.1" THEN "OUT_2-0.5" := FALSE; END_IF;
   #_w5 := #var[33] AND NOT "IN_7-0.1";
   IF #_w5 THEN
       #var[34] := TRUE;
       #var[33] := FALSE;
   END_IF;
   IF #var[34] THEN "OUT_2-0.0" := TRUE; END_IF;
   IF #var[34] AND NOT "IN_6-0.2" THEN "OUT_2-0.0" := FALSE; END_IF;
   #_w6 := #var[34] AND NOT "IN_6-0.2";
   IF #_w6 THEN
       #var[35] := TRUE;
       #var[34] := FALSE;
   END_IF;
   IF #var[35] THEN "OUT_2-0.5" := TRUE; END_IF;
   IF #var[35] AND NOT "IN_7-0.2" THEN "OUT_2-0.5" := FALSE; END_IF;
   #_w7 := #var[35] AND NOT "IN_7-0.2";
   IF #_w7 THEN
       #var[36] := TRUE;
       #var[35] := FALSE;
   END_IF;
   IF #var[36] THEN "OUT_2-0.4" := TRUE; END_IF;
   IF #var[36] AND NOT "IN_6-1.4" THEN "OUT_2-0.4" := FALSE; END_IF;
   #_w8 := #var[36] AND NOT "IN_6-1.4";
   IF #_w8 THEN
       #var[37] := TRUE;
       #var[36] := FALSE;
   END_IF;
   IF #var[37] THEN "OUT_2-0.6" := TRUE; END_IF;
   IF #var[37] AND NOT "IN_7-0.1" THEN
       "OUT_2-0.6" := FALSE;
       #var[37] := FALSE;
   END_IF;
END_REGION
END_FUNCTION_BLOCK

ORGANIZATION_BLOCK "Main"   // OB1, LAD, ProgramCycle
TITLE = "Main Program Sweep (Cycle)"
{ S7_Optimized_Access := 'TRUE' }
VERSION : 0.1
   VAR_INPUT
      Initial_Call : Bool;   // Initial call of this OB
      Remanence : Bool;   // =True, if remanent data are available
   END_VAR
BEGIN

REGION Network 1
   // Основая ветка: сервер контролера
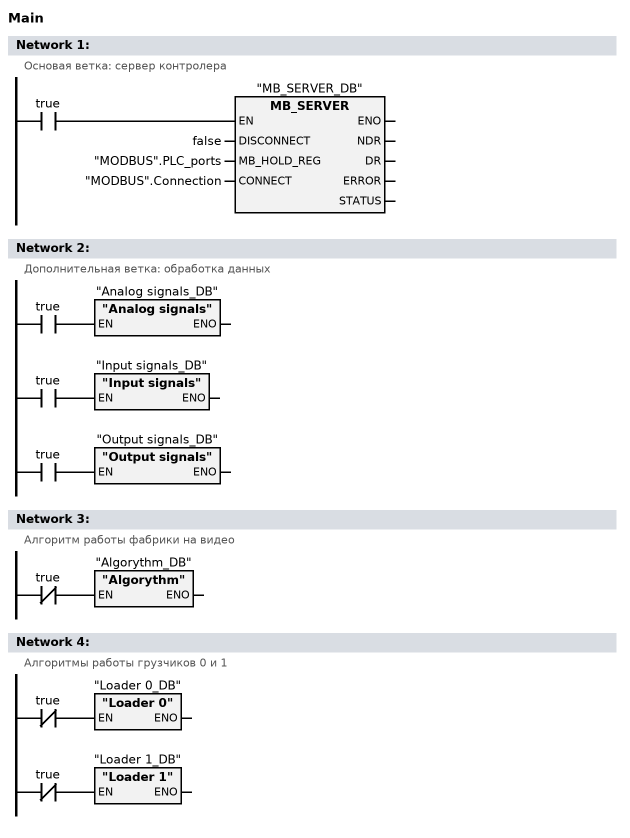
   IF true THEN
       "MB_SERVER_DB"(DISCONNECT := false, MB_HOLD_REG := "MODBUS".PLC_ports, CONNECT := "MODBUS".Connection);   // MB_SERVER
   END_IF;
END_REGION

REGION Network 2
   // Дополнительная ветка: обработка данных
   RUNG wire#powerrail
      Contact( true )
      "Analog signals_DB"()
   END_RUNG
   RUNG wire#powerrail
      Contact( true )
      "Input signals_DB"()
   END_RUNG
   RUNG wire#powerrail
      Contact( true )
      "Output signals_DB"()
   END_RUNG
   // the same network as SCL:
   IF true THEN
       "Analog signals_DB"();   // "Analog signals"
       "Input signals_DB"();   // "Input signals"
       "Output signals_DB"();   // "Output signals"
   END_IF;
END_REGION

REGION Network 3
   // Алгоритм работы фабрики на видео
   RUNG wire#powerrail
      I_Contact( true )
      "Algorythm_DB"()
   END_RUNG
   // the same network as SCL:
   IF NOT true THEN
       "Algorythm_DB"();   // "Algorythm"
   END_IF;
END_REGION

REGION Network 4
   // Алгоритмы работы грузчиков 0 и 1
   RUNG wire#powerrail
      I_Contact( true )
      "Loader 0_DB"()
   END_RUNG
   RUNG wire#powerrail
      I_Contact( true )
      "Loader 1_DB"()
   END_RUNG
   // the same network as SCL:
   IF NOT true THEN
       "Loader 0_DB"();   // "Loader 0"
       "Loader 1_DB"();   // "Loader 1"
   END_IF;
END_REGION
END_ORGANIZATION_BLOCK

// folder: Loaders

FUNCTION_BLOCK "Loader 0"   // FB5, LAD
{ S7_Optimized_Access := 'TRUE' }
VERSION : 0.1
BEGIN

REGION Network 1
   // Функция: ехать в 0 (1 ветка) или 1 (2 ветка) до нужного датчика (1-0.2 - 1-1.5)
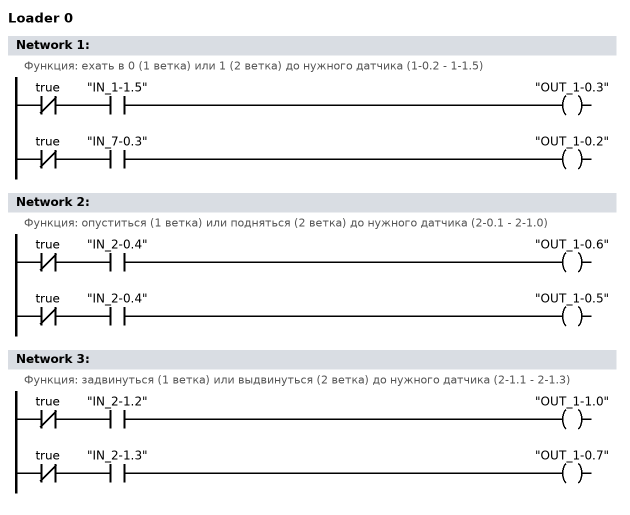
   RUNG wire#powerrail
      I_Contact( true )
      Contact( "IN_1-1.5" )
      Coil( "OUT_1-0.3" )
   END_RUNG
   RUNG wire#powerrail
      I_Contact( true )
      Contact( "IN_7-0.3" )
      Coil( "OUT_1-0.2" )
   END_RUNG
   // the same network as SCL:
   "OUT_1-0.3" := NOT true AND "IN_1-1.5";
   "OUT_1-0.2" := NOT true AND "IN_7-0.3";
END_REGION

REGION Network 2
   // Функция: опуститься (1 ветка) или подняться (2 ветка) до нужного датчика (2-0.1 - 2-1.0)
   RUNG wire#powerrail
      I_Contact( true )
      Contact( "IN_2-0.4" )
      Coil( "OUT_1-0.6" )
   END_RUNG
   RUNG wire#powerrail
      I_Contact( true )
      Contact( "IN_2-0.4" )
      Coil( "OUT_1-0.5" )
   END_RUNG
   // the same network as SCL:
   "OUT_1-0.6" := NOT true AND "IN_2-0.4";
   "OUT_1-0.5" := NOT true AND "IN_2-0.4";
END_REGION

REGION Network 3
   // Функция: задвинуться (1 ветка) или выдвинуться (2 ветка) до нужного датчика (2-1.1 - 2-1.3)
   RUNG wire#powerrail
      I_Contact( true )
      Contact( "IN_2-1.2" )
      Coil( "OUT_1-1.0" )
   END_RUNG
   RUNG wire#powerrail
      I_Contact( true )
      Contact( "IN_2-1.3" )
      Coil( "OUT_1-0.7" )
   END_RUNG
   // the same network as SCL:
   "OUT_1-1.0" := NOT true AND "IN_2-1.2";
   "OUT_1-0.7" := NOT true AND "IN_2-1.3";
END_REGION
END_FUNCTION_BLOCK

FUNCTION_BLOCK "Loader 1"   // FB6, LAD
{ S7_Optimized_Access := 'TRUE' }
VERSION : 0.1
BEGIN

REGION Network 1
   // Функция: ехать в 0 (1 ветка) или 1 (2 ветка) до нужного датчика (5-1.3 - 6-0.6)
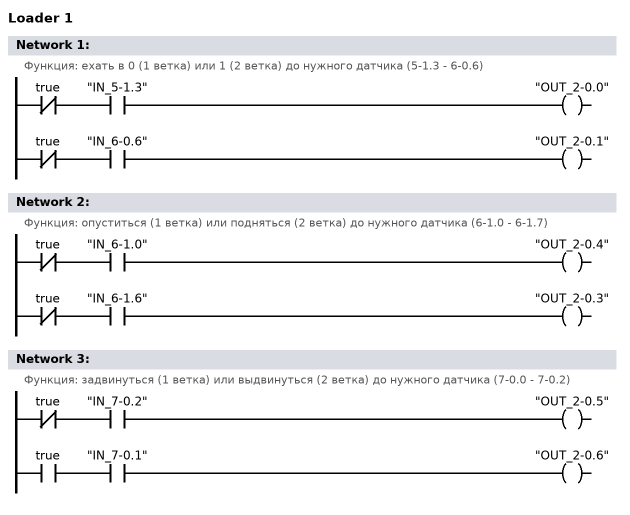
   RUNG wire#powerrail
      I_Contact( true )
      Contact( "IN_5-1.3" )
      Coil( "OUT_2-0.0" )
   END_RUNG
   RUNG wire#powerrail
      I_Contact( true )
      Contact( "IN_6-0.6" )
      Coil( "OUT_2-0.1" )
   END_RUNG
   // the same network as SCL:
   "OUT_2-0.0" := NOT true AND "IN_5-1.3";
   "OUT_2-0.1" := NOT true AND "IN_6-0.6";
END_REGION

REGION Network 2
   // Функция: опуститься (1 ветка) или подняться (2 ветка) до нужного датчика (6-1.0 - 6-1.7)
   RUNG wire#powerrail
      I_Contact( true )
      Contact( "IN_6-1.0" )
      Coil( "OUT_2-0.4" )
   END_RUNG
   RUNG wire#powerrail
      I_Contact( true )
      Contact( "IN_6-1.6" )
      Coil( "OUT_2-0.3" )
   END_RUNG
   // the same network as SCL:
   "OUT_2-0.4" := NOT true AND "IN_6-1.0";
   "OUT_2-0.3" := NOT true AND "IN_6-1.6";
END_REGION

REGION Network 3
   // Функция: задвинуться (1 ветка) или выдвинуться (2 ветка) до нужного датчика (7-0.0 - 7-0.2)
   RUNG wire#powerrail
      I_Contact( true )
      Contact( "IN_7-0.2" )
      Coil( "OUT_2-0.5" )
   END_RUNG
   RUNG wire#powerrail
      Contact( true )
      Contact( "IN_7-0.1" )
      Coil( "OUT_2-0.6" )
   END_RUNG
   // the same network as SCL:
   "OUT_2-0.5" := NOT true AND "IN_7-0.2";
   "OUT_2-0.6" := true AND "IN_7-0.1";
END_REGION
END_FUNCTION_BLOCK

// folder: PLC signals

FUNCTION_BLOCK "Analog signals"   // FB1, LAD
{ S7_Optimized_Access := 'TRUE' }
VERSION : 0.1
   VAR
      var : Array[0..4] of Bool;
   END_VAR
   VAR_TEMP
      i : Bool;
   END_VAR
BEGIN

REGION Network 1
   // Аналоговые входы блока Siemens S7-1200
   // 1 - желтый, 2 - синий, 3 - зеленый, 4 - фиолетовый (0 - черный)
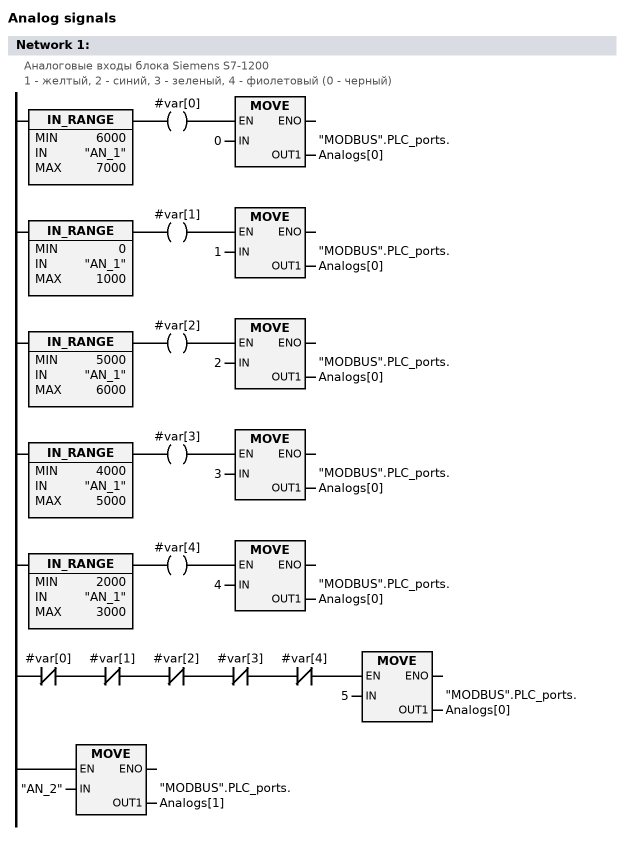
   RUNG wire#powerrail
      { S7_Templates := "SrcType := Int" } InRange(min := 6000, in := "AN_1", max := 7000)
      Coil( #var[0] )
      Move(in := 0, out1 => "MODBUS".PLC_ports.Analogs[0])
   END_RUNG
   RUNG wire#powerrail
      { S7_Templates := "SrcType := Int" } InRange(min := 0, in := "AN_1", max := 1000)
      Coil( #var[1] )
      Move(in := 1, out1 => "MODBUS".PLC_ports.Analogs[0])
   END_RUNG
   RUNG wire#powerrail
      { S7_Templates := "SrcType := Int" } InRange(min := 5000, in := "AN_1", max := 6000)
      Coil( #var[2] )
      Move(in := 2, out1 => "MODBUS".PLC_ports.Analogs[0])
   END_RUNG
   RUNG wire#powerrail
      { S7_Templates := "SrcType := Int" } InRange(min := 4000, in := "AN_1", max := 5000)
      Coil( #var[3] )
      Move(in := 3, out1 => "MODBUS".PLC_ports.Analogs[0])
   END_RUNG
   RUNG wire#powerrail
      { S7_Templates := "SrcType := Int" } InRange(min := 2000, in := "AN_1", max := 3000)
      Coil( #var[4] )
      Move(in := 4, out1 => "MODBUS".PLC_ports.Analogs[0])
   END_RUNG
   RUNG wire#powerrail
      I_Contact( #var[0] )
      I_Contact( #var[1] )
      I_Contact( #var[2] )
      I_Contact( #var[3] )
      I_Contact( #var[4] )
      Move(in := 5, out1 => "MODBUS".PLC_ports.Analogs[0])
   END_RUNG
   RUNG wire#powerrail
      Move(in := "AN_2", out1 => "MODBUS".PLC_ports.Analogs[1])
   END_RUNG
   // the same network as SCL:
   #var[0] := (6000 <= "AN_1") AND ("AN_1" <= 7000);
   IF (6000 <= "AN_1") AND ("AN_1" <= 7000) THEN "MODBUS".PLC_ports.Analogs[0] := 0; END_IF;
   #var[1] := (0 <= "AN_1") AND ("AN_1" <= 1000);
   IF (0 <= "AN_1") AND ("AN_1" <= 1000) THEN "MODBUS".PLC_ports.Analogs[0] := 1; END_IF;
   #var[2] := (5000 <= "AN_1") AND ("AN_1" <= 6000);
   IF (5000 <= "AN_1") AND ("AN_1" <= 6000) THEN "MODBUS".PLC_ports.Analogs[0] := 2; END_IF;
   #var[3] := (4000 <= "AN_1") AND ("AN_1" <= 5000);
   IF (4000 <= "AN_1") AND ("AN_1" <= 5000) THEN "MODBUS".PLC_ports.Analogs[0] := 3; END_IF;
   #var[4] := (2000 <= "AN_1") AND ("AN_1" <= 3000);
   IF (2000 <= "AN_1") AND ("AN_1" <= 3000) THEN "MODBUS".PLC_ports.Analogs[0] := 4; END_IF;
   IF NOT #var[0] AND NOT #var[1] AND NOT #var[2] AND NOT #var[3] AND NOT #var[4] THEN
       "MODBUS".PLC_ports.Analogs[0] := 5;
   END_IF;
   "MODBUS".PLC_ports.Analogs[1] := "AN_2";
END_REGION
END_FUNCTION_BLOCK

FUNCTION_BLOCK "Input signals"   // FB2, LAD
{ S7_Optimized_Access := 'TRUE' }
VERSION : 0.1
BEGIN

REGION Network 1
   // Входы 1 блока, Siemens S7-1200
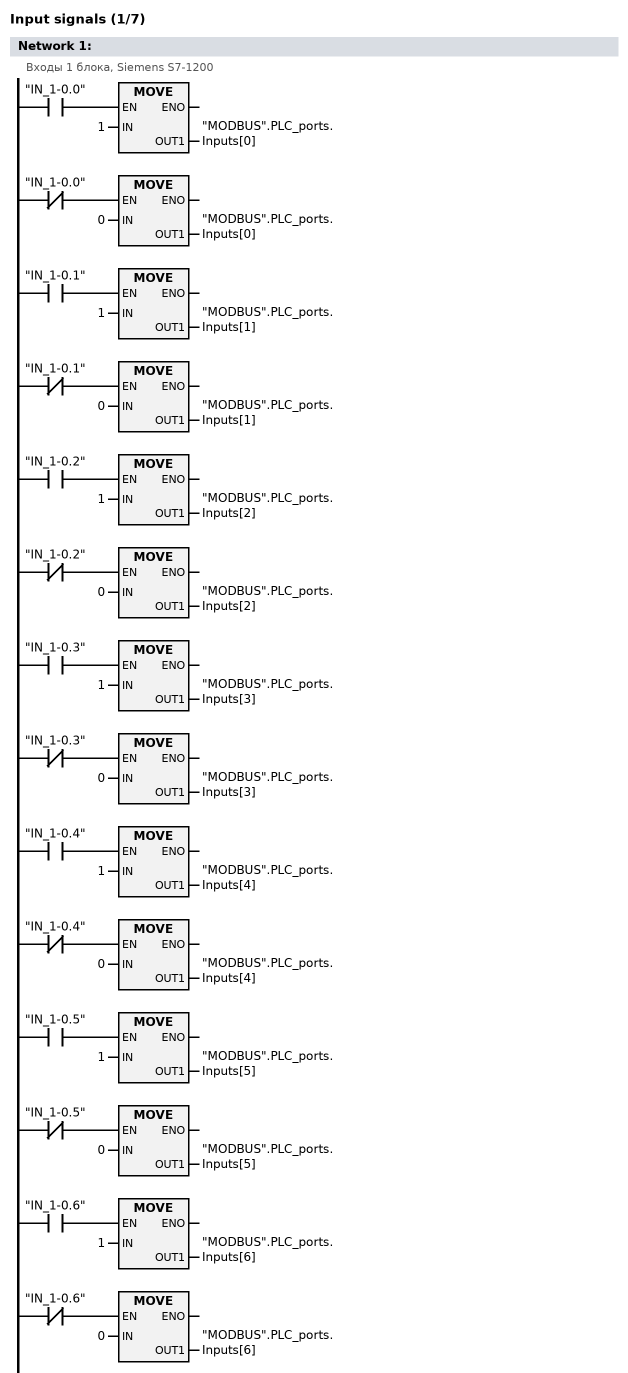
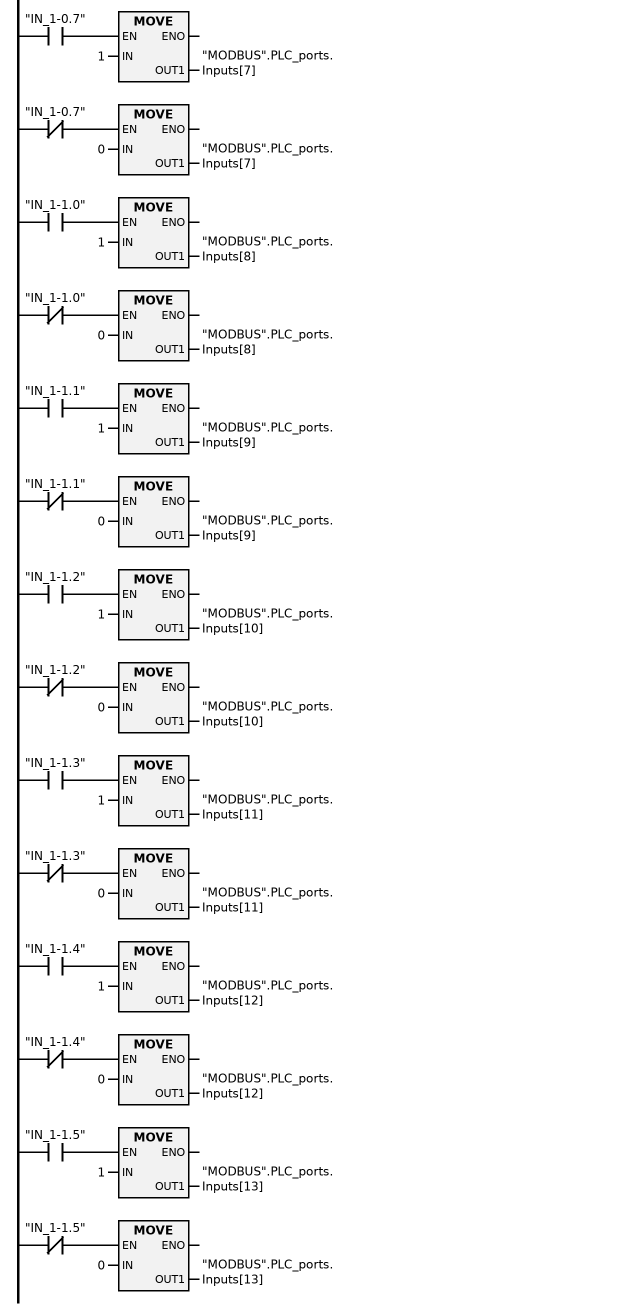
   RUNG wire#powerrail
      Contact( "IN_1-0.0" )
      Move(in := 1, out1 => "MODBUS".PLC_ports.Inputs[0])
   END_RUNG
   RUNG wire#powerrail
      I_Contact( "IN_1-0.0" )
      Move(in := 0, out1 => "MODBUS".PLC_ports.Inputs[0])
   END_RUNG
   RUNG wire#powerrail
      Contact( "IN_1-0.1" )
      Move(in := 1, out1 => "MODBUS".PLC_ports.Inputs[1])
   END_RUNG
   RUNG wire#powerrail
      I_Contact( "IN_1-0.1" )
      Move(in := 0, out1 => "MODBUS".PLC_ports.Inputs[1])
   END_RUNG
   RUNG wire#powerrail
      Contact( "IN_1-0.2" )
      Move(in := 1, out1 => "MODBUS".PLC_ports.Inputs[2])
   END_RUNG
   RUNG wire#powerrail
      I_Contact( "IN_1-0.2" )
      Move(in := 0, out1 => "MODBUS".PLC_ports.Inputs[2])
   END_RUNG
   RUNG wire#powerrail
      Contact( "IN_1-0.3" )
      Move(in := 1, out1 => "MODBUS".PLC_ports.Inputs[3])
   END_RUNG
   RUNG wire#powerrail
      I_Contact( "IN_1-0.3" )
      Move(in := 0, out1 => "MODBUS".PLC_ports.Inputs[3])
   END_RUNG
   RUNG wire#powerrail
      Contact( "IN_1-0.4" )
      Move(in := 1, out1 => "MODBUS".PLC_ports.Inputs[4])
   END_RUNG
   RUNG wire#powerrail
      I_Contact( "IN_1-0.4" )
      Move(in := 0, out1 => "MODBUS".PLC_ports.Inputs[4])
   END_RUNG
   RUNG wire#powerrail
      Contact( "IN_1-0.5" )
      Move(in := 1, out1 => "MODBUS".PLC_ports.Inputs[5])
   END_RUNG
   RUNG wire#powerrail
      I_Contact( "IN_1-0.5" )
      Move(in := 0, out1 => "MODBUS".PLC_ports.Inputs[5])
   END_RUNG
   RUNG wire#powerrail
      Contact( "IN_1-0.6" )
      Move(in := 1, out1 => "MODBUS".PLC_ports.Inputs[6])
   END_RUNG
   RUNG wire#powerrail
      I_Contact( "IN_1-0.6" )
      Move(in := 0, out1 => "MODBUS".PLC_ports.Inputs[6])
   END_RUNG
   RUNG wire#powerrail
      Contact( "IN_1-0.7" )
      Move(in := 1, out1 => "MODBUS".PLC_ports.Inputs[7])
   END_RUNG
   RUNG wire#powerrail
      I_Contact( "IN_1-0.7" )
      Move(in := 0, out1 => "MODBUS".PLC_ports.Inputs[7])
   END_RUNG
   RUNG wire#powerrail
      Contact( "IN_1-1.0" )
      Move(in := 1, out1 => "MODBUS".PLC_ports.Inputs[8])
   END_RUNG
   RUNG wire#powerrail
      I_Contact( "IN_1-1.0" )
      Move(in := 0, out1 => "MODBUS".PLC_ports.Inputs[8])
   END_RUNG
   RUNG wire#powerrail
      Contact( "IN_1-1.1" )
      Move(in := 1, out1 => "MODBUS".PLC_ports.Inputs[9])
   END_RUNG
   RUNG wire#powerrail
      I_Contact( "IN_1-1.1" )
      Move(in := 0, out1 => "MODBUS".PLC_ports.Inputs[9])
   END_RUNG
   RUNG wire#powerrail
      Contact( "IN_1-1.2" )
      Move(in := 1, out1 => "MODBUS".PLC_ports.Inputs[10])
   END_RUNG
   RUNG wire#powerrail
      I_Contact( "IN_1-1.2" )
      Move(in := 0, out1 => "MODBUS".PLC_ports.Inputs[10])
   END_RUNG
   RUNG wire#powerrail
      Contact( "IN_1-1.3" )
      Move(in := 1, out1 => "MODBUS".PLC_ports.Inputs[11])
   END_RUNG
   RUNG wire#powerrail
      I_Contact( "IN_1-1.3" )
      Move(in := 0, out1 => "MODBUS".PLC_ports.Inputs[11])
   END_RUNG
   RUNG wire#powerrail
      Contact( "IN_1-1.4" )
      Move(in := 1, out1 => "MODBUS".PLC_ports.Inputs[12])
   END_RUNG
   RUNG wire#powerrail
      I_Contact( "IN_1-1.4" )
      Move(in := 0, out1 => "MODBUS".PLC_ports.Inputs[12])
   END_RUNG
   RUNG wire#powerrail
      Contact( "IN_1-1.5" )
      Move(in := 1, out1 => "MODBUS".PLC_ports.Inputs[13])
   END_RUNG
   RUNG wire#powerrail
      I_Contact( "IN_1-1.5" )
      Move(in := 0, out1 => "MODBUS".PLC_ports.Inputs[13])
   END_RUNG
   // the same network as SCL:
   IF "IN_1-0.0" THEN "MODBUS".PLC_ports.Inputs[0] := 1; END_IF;
   IF NOT "IN_1-0.0" THEN "MODBUS".PLC_ports.Inputs[0] := 0; END_IF;
   IF "IN_1-0.1" THEN "MODBUS".PLC_ports.Inputs[1] := 1; END_IF;
   IF NOT "IN_1-0.1" THEN "MODBUS".PLC_ports.Inputs[1] := 0; END_IF;
   IF "IN_1-0.2" THEN "MODBUS".PLC_ports.Inputs[2] := 1; END_IF;
   IF NOT "IN_1-0.2" THEN "MODBUS".PLC_ports.Inputs[2] := 0; END_IF;
   IF "IN_1-0.3" THEN "MODBUS".PLC_ports.Inputs[3] := 1; END_IF;
   IF NOT "IN_1-0.3" THEN "MODBUS".PLC_ports.Inputs[3] := 0; END_IF;
   IF "IN_1-0.4" THEN "MODBUS".PLC_ports.Inputs[4] := 1; END_IF;
   IF NOT "IN_1-0.4" THEN "MODBUS".PLC_ports.Inputs[4] := 0; END_IF;
   IF "IN_1-0.5" THEN "MODBUS".PLC_ports.Inputs[5] := 1; END_IF;
   IF NOT "IN_1-0.5" THEN "MODBUS".PLC_ports.Inputs[5] := 0; END_IF;
   IF "IN_1-0.6" THEN "MODBUS".PLC_ports.Inputs[6] := 1; END_IF;
   IF NOT "IN_1-0.6" THEN "MODBUS".PLC_ports.Inputs[6] := 0; END_IF;
   IF "IN_1-0.7" THEN "MODBUS".PLC_ports.Inputs[7] := 1; END_IF;
   IF NOT "IN_1-0.7" THEN "MODBUS".PLC_ports.Inputs[7] := 0; END_IF;
   IF "IN_1-1.0" THEN "MODBUS".PLC_ports.Inputs[8] := 1; END_IF;
   IF NOT "IN_1-1.0" THEN "MODBUS".PLC_ports.Inputs[8] := 0; END_IF;
   IF "IN_1-1.1" THEN "MODBUS".PLC_ports.Inputs[9] := 1; END_IF;
   IF NOT "IN_1-1.1" THEN "MODBUS".PLC_ports.Inputs[9] := 0; END_IF;
   IF "IN_1-1.2" THEN "MODBUS".PLC_ports.Inputs[10] := 1; END_IF;
   IF NOT "IN_1-1.2" THEN "MODBUS".PLC_ports.Inputs[10] := 0; END_IF;
   IF "IN_1-1.3" THEN "MODBUS".PLC_ports.Inputs[11] := 1; END_IF;
   IF NOT "IN_1-1.3" THEN "MODBUS".PLC_ports.Inputs[11] := 0; END_IF;
   IF "IN_1-1.4" THEN "MODBUS".PLC_ports.Inputs[12] := 1; END_IF;
   IF NOT "IN_1-1.4" THEN "MODBUS".PLC_ports.Inputs[12] := 0; END_IF;
   IF "IN_1-1.5" THEN "MODBUS".PLC_ports.Inputs[13] := 1; END_IF;
   IF NOT "IN_1-1.5" THEN "MODBUS".PLC_ports.Inputs[13] := 0; END_IF;
END_REGION

REGION Network 2
   // Входы 2 блока, Siemens SM-1223
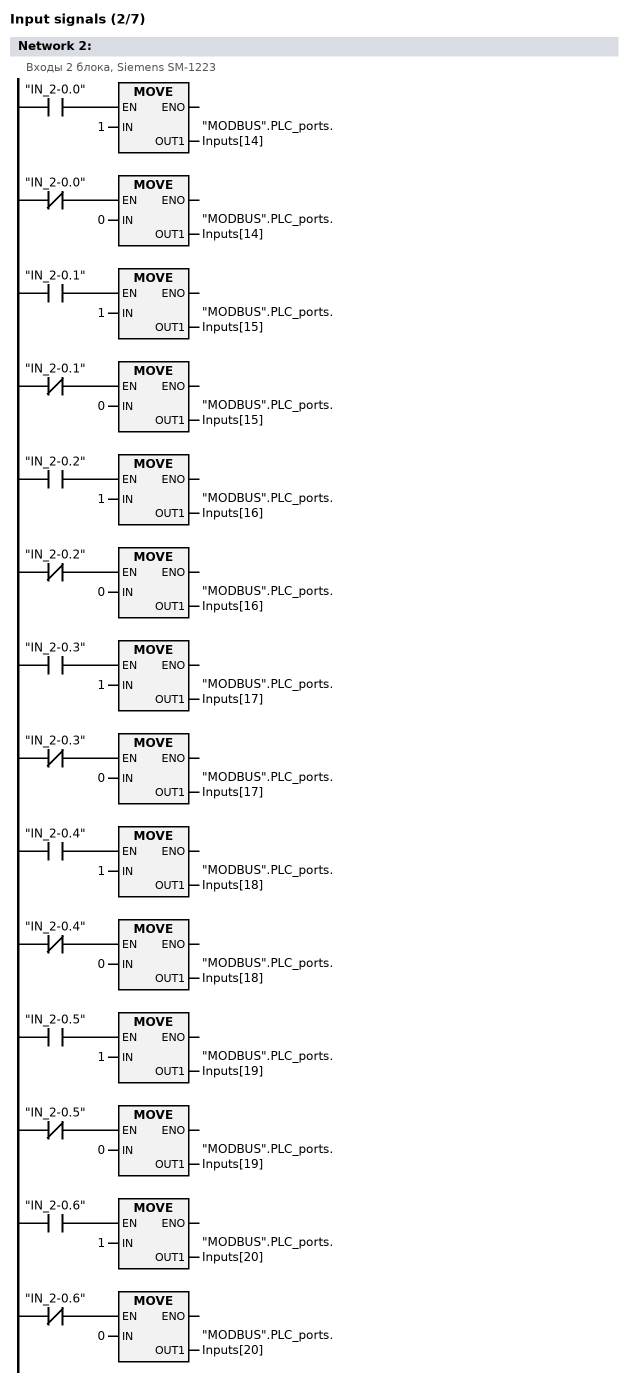
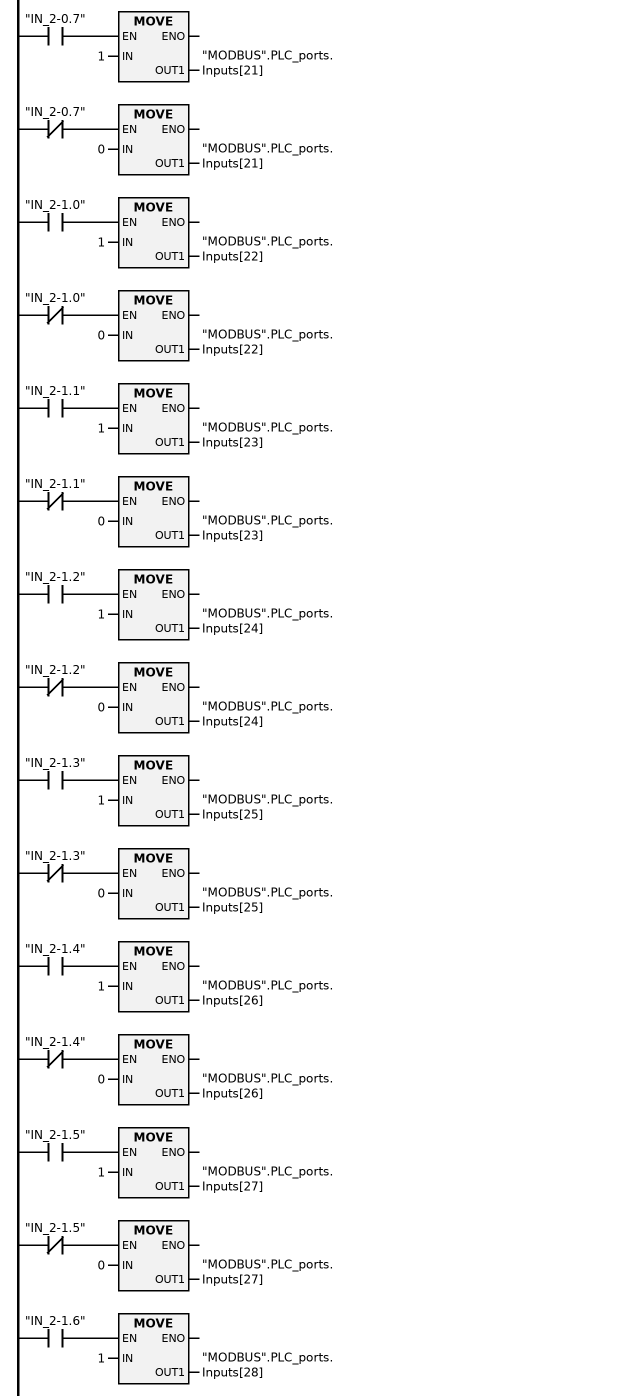
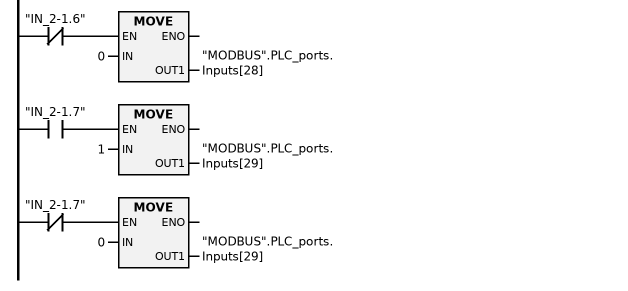
   RUNG wire#powerrail
      Contact( "IN_2-0.0" )
      Move(in := 1, out1 => "MODBUS".PLC_ports.Inputs[14])
   END_RUNG
   RUNG wire#powerrail
      I_Contact( "IN_2-0.0" )
      Move(in := 0, out1 => "MODBUS".PLC_ports.Inputs[14])
   END_RUNG
   RUNG wire#powerrail
      Contact( "IN_2-0.1" )
      Move(in := 1, out1 => "MODBUS".PLC_ports.Inputs[15])
   END_RUNG
   RUNG wire#powerrail
      I_Contact( "IN_2-0.1" )
      Move(in := 0, out1 => "MODBUS".PLC_ports.Inputs[15])
   END_RUNG
   RUNG wire#powerrail
      Contact( "IN_2-0.2" )
      Move(in := 1, out1 => "MODBUS".PLC_ports.Inputs[16])
   END_RUNG
   RUNG wire#powerrail
      I_Contact( "IN_2-0.2" )
      Move(in := 0, out1 => "MODBUS".PLC_ports.Inputs[16])
   END_RUNG
   RUNG wire#powerrail
      Contact( "IN_2-0.3" )
      Move(in := 1, out1 => "MODBUS".PLC_ports.Inputs[17])
   END_RUNG
   RUNG wire#powerrail
      I_Contact( "IN_2-0.3" )
      Move(in := 0, out1 => "MODBUS".PLC_ports.Inputs[17])
   END_RUNG
   RUNG wire#powerrail
      Contact( "IN_2-0.4" )
      Move(in := 1, out1 => "MODBUS".PLC_ports.Inputs[18])
   END_RUNG
   RUNG wire#powerrail
      I_Contact( "IN_2-0.4" )
      Move(in := 0, out1 => "MODBUS".PLC_ports.Inputs[18])
   END_RUNG
   RUNG wire#powerrail
      Contact( "IN_2-0.5" )
      Move(in := 1, out1 => "MODBUS".PLC_ports.Inputs[19])
   END_RUNG
   RUNG wire#powerrail
      I_Contact( "IN_2-0.5" )
      Move(in := 0, out1 => "MODBUS".PLC_ports.Inputs[19])
   END_RUNG
   RUNG wire#powerrail
      Contact( "IN_2-0.6" )
      Move(in := 1, out1 => "MODBUS".PLC_ports.Inputs[20])
   END_RUNG
   RUNG wire#powerrail
      I_Contact( "IN_2-0.6" )
      Move(in := 0, out1 => "MODBUS".PLC_ports.Inputs[20])
   END_RUNG
   RUNG wire#powerrail
      Contact( "IN_2-0.7" )
      Move(in := 1, out1 => "MODBUS".PLC_ports.Inputs[21])
   END_RUNG
   RUNG wire#powerrail
      I_Contact( "IN_2-0.7" )
      Move(in := 0, out1 => "MODBUS".PLC_ports.Inputs[21])
   END_RUNG
   RUNG wire#powerrail
      Contact( "IN_2-1.0" )
      Move(in := 1, out1 => "MODBUS".PLC_ports.Inputs[22])
   END_RUNG
   RUNG wire#powerrail
      I_Contact( "IN_2-1.0" )
      Move(in := 0, out1 => "MODBUS".PLC_ports.Inputs[22])
   END_RUNG
   RUNG wire#powerrail
      Contact( "IN_2-1.1" )
      Move(in := 1, out1 => "MODBUS".PLC_ports.Inputs[23])
   END_RUNG
   RUNG wire#powerrail
      I_Contact( "IN_2-1.1" )
      Move(in := 0, out1 => "MODBUS".PLC_ports.Inputs[23])
   END_RUNG
   RUNG wire#powerrail
      Contact( "IN_2-1.2" )
      Move(in := 1, out1 => "MODBUS".PLC_ports.Inputs[24])
   END_RUNG
   RUNG wire#powerrail
      I_Contact( "IN_2-1.2" )
      Move(in := 0, out1 => "MODBUS".PLC_ports.Inputs[24])
   END_RUNG
   RUNG wire#powerrail
      Contact( "IN_2-1.3" )
      Move(in := 1, out1 => "MODBUS".PLC_ports.Inputs[25])
   END_RUNG
   RUNG wire#powerrail
      I_Contact( "IN_2-1.3" )
      Move(in := 0, out1 => "MODBUS".PLC_ports.Inputs[25])
   END_RUNG
   RUNG wire#powerrail
      Contact( "IN_2-1.4" )
      Move(in := 1, out1 => "MODBUS".PLC_ports.Inputs[26])
   END_RUNG
   RUNG wire#powerrail
      I_Contact( "IN_2-1.4" )
      Move(in := 0, out1 => "MODBUS".PLC_ports.Inputs[26])
   END_RUNG
   RUNG wire#powerrail
      Contact( "IN_2-1.5" )
      Move(in := 1, out1 => "MODBUS".PLC_ports.Inputs[27])
   END_RUNG
   RUNG wire#powerrail
      I_Contact( "IN_2-1.5" )
      Move(in := 0, out1 => "MODBUS".PLC_ports.Inputs[27])
   END_RUNG
   RUNG wire#powerrail
      Contact( "IN_2-1.6" )
      Move(in := 1, out1 => "MODBUS".PLC_ports.Inputs[28])
   END_RUNG
   RUNG wire#powerrail
      I_Contact( "IN_2-1.6" )
      Move(in := 0, out1 => "MODBUS".PLC_ports.Inputs[28])
   END_RUNG
   RUNG wire#powerrail
      Contact( "IN_2-1.7" )
      Move(in := 1, out1 => "MODBUS".PLC_ports.Inputs[29])
   END_RUNG
   RUNG wire#powerrail
      I_Contact( "IN_2-1.7" )
      Move(in := 0, out1 => "MODBUS".PLC_ports.Inputs[29])
   END_RUNG
   // the same network as SCL:
   IF "IN_2-0.0" THEN "MODBUS".PLC_ports.Inputs[14] := 1; END_IF;
   IF NOT "IN_2-0.0" THEN "MODBUS".PLC_ports.Inputs[14] := 0; END_IF;
   IF "IN_2-0.1" THEN "MODBUS".PLC_ports.Inputs[15] := 1; END_IF;
   IF NOT "IN_2-0.1" THEN "MODBUS".PLC_ports.Inputs[15] := 0; END_IF;
   IF "IN_2-0.2" THEN "MODBUS".PLC_ports.Inputs[16] := 1; END_IF;
   IF NOT "IN_2-0.2" THEN "MODBUS".PLC_ports.Inputs[16] := 0; END_IF;
   IF "IN_2-0.3" THEN "MODBUS".PLC_ports.Inputs[17] := 1; END_IF;
   IF NOT "IN_2-0.3" THEN "MODBUS".PLC_ports.Inputs[17] := 0; END_IF;
   IF "IN_2-0.4" THEN "MODBUS".PLC_ports.Inputs[18] := 1; END_IF;
   IF NOT "IN_2-0.4" THEN "MODBUS".PLC_ports.Inputs[18] := 0; END_IF;
   IF "IN_2-0.5" THEN "MODBUS".PLC_ports.Inputs[19] := 1; END_IF;
   IF NOT "IN_2-0.5" THEN "MODBUS".PLC_ports.Inputs[19] := 0; END_IF;
   IF "IN_2-0.6" THEN "MODBUS".PLC_ports.Inputs[20] := 1; END_IF;
   IF NOT "IN_2-0.6" THEN "MODBUS".PLC_ports.Inputs[20] := 0; END_IF;
   IF "IN_2-0.7" THEN "MODBUS".PLC_ports.Inputs[21] := 1; END_IF;
   IF NOT "IN_2-0.7" THEN "MODBUS".PLC_ports.Inputs[21] := 0; END_IF;
   IF "IN_2-1.0" THEN "MODBUS".PLC_ports.Inputs[22] := 1; END_IF;
   IF NOT "IN_2-1.0" THEN "MODBUS".PLC_ports.Inputs[22] := 0; END_IF;
   IF "IN_2-1.1" THEN "MODBUS".PLC_ports.Inputs[23] := 1; END_IF;
   IF NOT "IN_2-1.1" THEN "MODBUS".PLC_ports.Inputs[23] := 0; END_IF;
   IF "IN_2-1.2" THEN "MODBUS".PLC_ports.Inputs[24] := 1; END_IF;
   IF NOT "IN_2-1.2" THEN "MODBUS".PLC_ports.Inputs[24] := 0; END_IF;
   IF "IN_2-1.3" THEN "MODBUS".PLC_ports.Inputs[25] := 1; END_IF;
   IF NOT "IN_2-1.3" THEN "MODBUS".PLC_ports.Inputs[25] := 0; END_IF;
   IF "IN_2-1.4" THEN "MODBUS".PLC_ports.Inputs[26] := 1; END_IF;
   IF NOT "IN_2-1.4" THEN "MODBUS".PLC_ports.Inputs[26] := 0; END_IF;
   IF "IN_2-1.5" THEN "MODBUS".PLC_ports.Inputs[27] := 1; END_IF;
   IF NOT "IN_2-1.5" THEN "MODBUS".PLC_ports.Inputs[27] := 0; END_IF;
   IF "IN_2-1.6" THEN "MODBUS".PLC_ports.Inputs[28] := 1; END_IF;
   IF NOT "IN_2-1.6" THEN "MODBUS".PLC_ports.Inputs[28] := 0; END_IF;
   IF "IN_2-1.7" THEN "MODBUS".PLC_ports.Inputs[29] := 1; END_IF;
   IF NOT "IN_2-1.7" THEN "MODBUS".PLC_ports.Inputs[29] := 0; END_IF;
END_REGION

REGION Network 3
   // Входы 3 блока, Siemens SM-1223
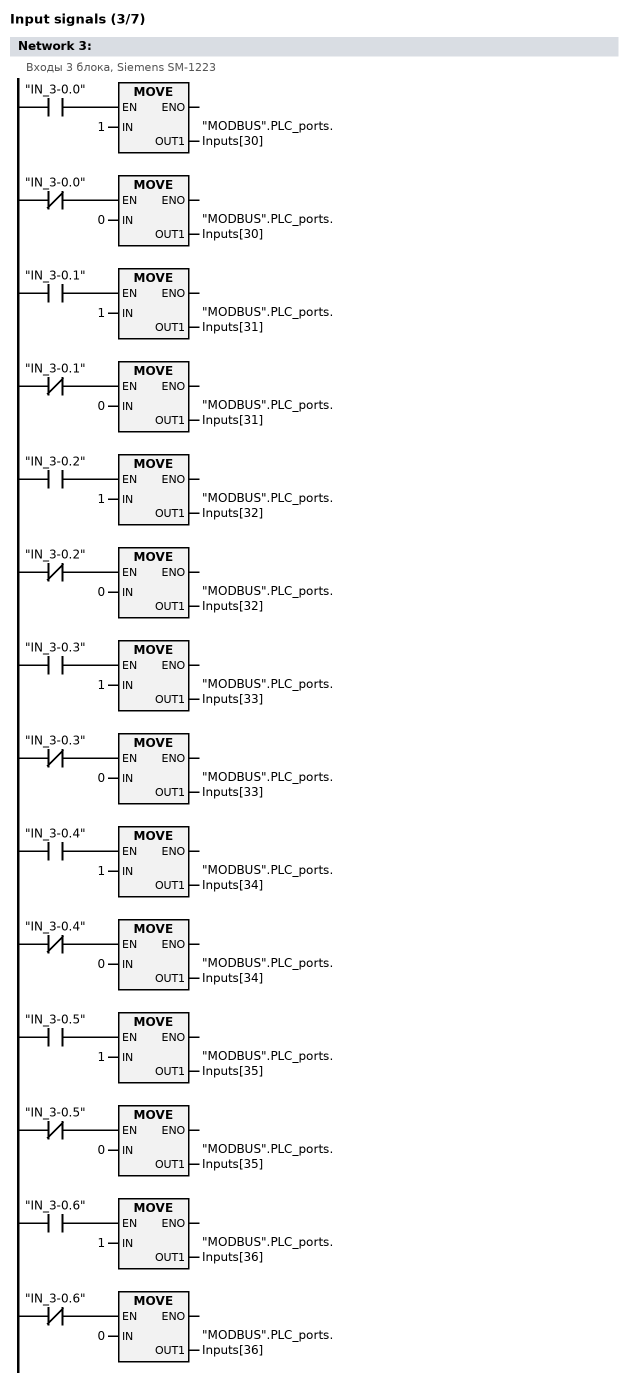
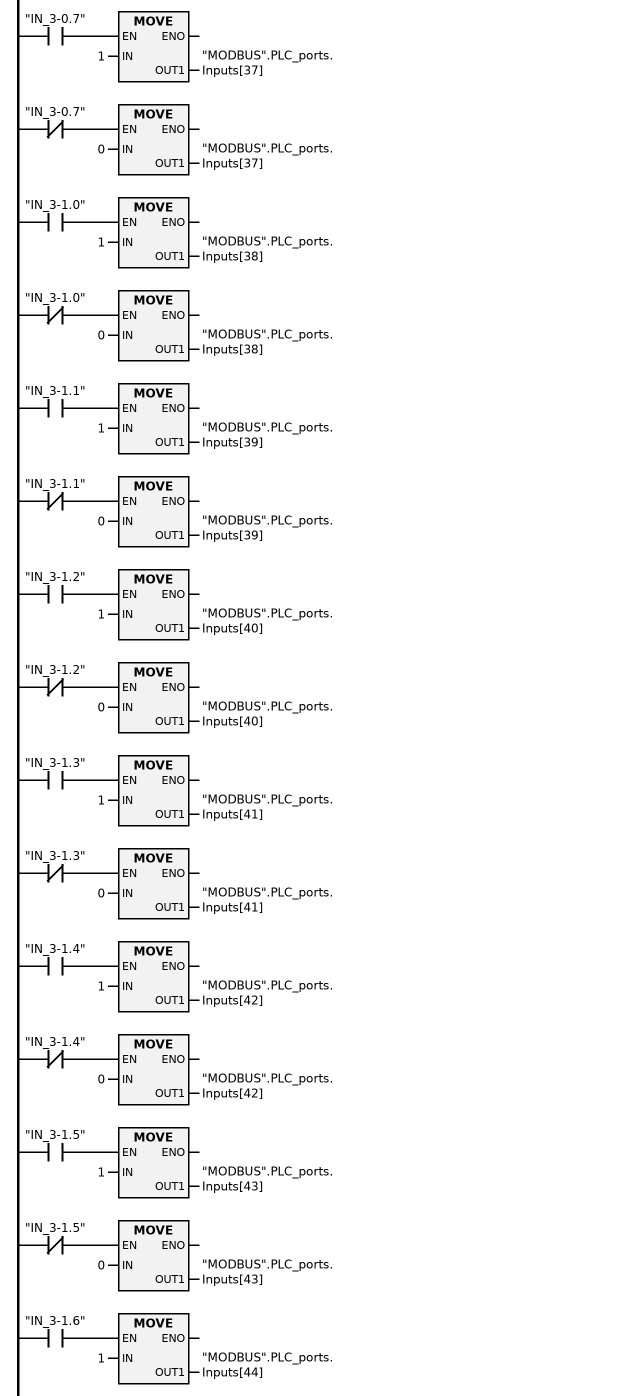
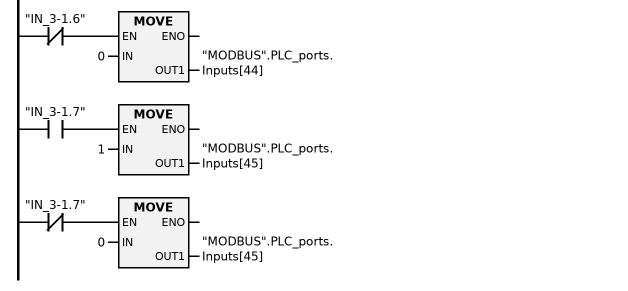
   RUNG wire#powerrail
      Contact( "IN_3-0.0" )
      Move(in := 1, out1 => "MODBUS".PLC_ports.Inputs[30])
   END_RUNG
   RUNG wire#powerrail
      I_Contact( "IN_3-0.0" )
      Move(in := 0, out1 => "MODBUS".PLC_ports.Inputs[30])
   END_RUNG
   RUNG wire#powerrail
      Contact( "IN_3-0.1" )
      Move(in := 1, out1 => "MODBUS".PLC_ports.Inputs[31])
   END_RUNG
   RUNG wire#powerrail
      I_Contact( "IN_3-0.1" )
      Move(in := 0, out1 => "MODBUS".PLC_ports.Inputs[31])
   END_RUNG
   RUNG wire#powerrail
      Contact( "IN_3-0.2" )
      Move(in := 1, out1 => "MODBUS".PLC_ports.Inputs[32])
   END_RUNG
   RUNG wire#powerrail
      I_Contact( "IN_3-0.2" )
      Move(in := 0, out1 => "MODBUS".PLC_ports.Inputs[32])
   END_RUNG
   RUNG wire#powerrail
      Contact( "IN_3-0.3" )
      Move(in := 1, out1 => "MODBUS".PLC_ports.Inputs[33])
   END_RUNG
   RUNG wire#powerrail
      I_Contact( "IN_3-0.3" )
      Move(in := 0, out1 => "MODBUS".PLC_ports.Inputs[33])
   END_RUNG
   RUNG wire#powerrail
      Contact( "IN_3-0.4" )
      Move(in := 1, out1 => "MODBUS".PLC_ports.Inputs[34])
   END_RUNG
   RUNG wire#powerrail
      I_Contact( "IN_3-0.4" )
      Move(in := 0, out1 => "MODBUS".PLC_ports.Inputs[34])
   END_RUNG
   RUNG wire#powerrail
      Contact( "IN_3-0.5" )
      Move(in := 1, out1 => "MODBUS".PLC_ports.Inputs[35])
   END_RUNG
   RUNG wire#powerrail
      I_Contact( "IN_3-0.5" )
      Move(in := 0, out1 => "MODBUS".PLC_ports.Inputs[35])
   END_RUNG
   RUNG wire#powerrail
      Contact( "IN_3-0.6" )
      Move(in := 1, out1 => "MODBUS".PLC_ports.Inputs[36])
   END_RUNG
   RUNG wire#powerrail
      I_Contact( "IN_3-0.6" )
      Move(in := 0, out1 => "MODBUS".PLC_ports.Inputs[36])
   END_RUNG
   RUNG wire#powerrail
      Contact( "IN_3-0.7" )
      Move(in := 1, out1 => "MODBUS".PLC_ports.Inputs[37])
   END_RUNG
   RUNG wire#powerrail
      I_Contact( "IN_3-0.7" )
      Move(in := 0, out1 => "MODBUS".PLC_ports.Inputs[37])
   END_RUNG
   RUNG wire#powerrail
      Contact( "IN_3-1.0" )
      Move(in := 1, out1 => "MODBUS".PLC_ports.Inputs[38])
   END_RUNG
   RUNG wire#powerrail
      I_Contact( "IN_3-1.0" )
      Move(in := 0, out1 => "MODBUS".PLC_ports.Inputs[38])
   END_RUNG
   RUNG wire#powerrail
      Contact( "IN_3-1.1" )
      Move(in := 1, out1 => "MODBUS".PLC_ports.Inputs[39])
   END_RUNG
   RUNG wire#powerrail
      I_Contact( "IN_3-1.1" )
      Move(in := 0, out1 => "MODBUS".PLC_ports.Inputs[39])
   END_RUNG
   RUNG wire#powerrail
      Contact( "IN_3-1.2" )
      Move(in := 1, out1 => "MODBUS".PLC_ports.Inputs[40])
   END_RUNG
   RUNG wire#powerrail
      I_Contact( "IN_3-1.2" )
      Move(in := 0, out1 => "MODBUS".PLC_ports.Inputs[40])
   END_RUNG
   RUNG wire#powerrail
      Contact( "IN_3-1.3" )
      Move(in := 1, out1 => "MODBUS".PLC_ports.Inputs[41])
   END_RUNG
   RUNG wire#powerrail
      I_Contact( "IN_3-1.3" )
      Move(in := 0, out1 => "MODBUS".PLC_ports.Inputs[41])
   END_RUNG
   RUNG wire#powerrail
      Contact( "IN_3-1.4" )
      Move(in := 1, out1 => "MODBUS".PLC_ports.Inputs[42])
   END_RUNG
   RUNG wire#powerrail
      I_Contact( "IN_3-1.4" )
      Move(in := 0, out1 => "MODBUS".PLC_ports.Inputs[42])
   END_RUNG
   RUNG wire#powerrail
      Contact( "IN_3-1.5" )
      Move(in := 1, out1 => "MODBUS".PLC_ports.Inputs[43])
   END_RUNG
   RUNG wire#powerrail
      I_Contact( "IN_3-1.5" )
      Move(in := 0, out1 => "MODBUS".PLC_ports.Inputs[43])
   END_RUNG
   RUNG wire#powerrail
      Contact( "IN_3-1.6" )
      Move(in := 1, out1 => "MODBUS".PLC_ports.Inputs[44])
   END_RUNG
   RUNG wire#powerrail
      I_Contact( "IN_3-1.6" )
      Move(in := 0, out1 => "MODBUS".PLC_ports.Inputs[44])
   END_RUNG
   RUNG wire#powerrail
      Contact( "IN_3-1.7" )
      Move(in := 1, out1 => "MODBUS".PLC_ports.Inputs[45])
   END_RUNG
   RUNG wire#powerrail
      I_Contact( "IN_3-1.7" )
      Move(in := 0, out1 => "MODBUS".PLC_ports.Inputs[45])
   END_RUNG
   // the same network as SCL:
   IF "IN_3-0.0" THEN "MODBUS".PLC_ports.Inputs[30] := 1; END_IF;
   IF NOT "IN_3-0.0" THEN "MODBUS".PLC_ports.Inputs[30] := 0; END_IF;
   IF "IN_3-0.1" THEN "MODBUS".PLC_ports.Inputs[31] := 1; END_IF;
   IF NOT "IN_3-0.1" THEN "MODBUS".PLC_ports.Inputs[31] := 0; END_IF;
   IF "IN_3-0.2" THEN "MODBUS".PLC_ports.Inputs[32] := 1; END_IF;
   IF NOT "IN_3-0.2" THEN "MODBUS".PLC_ports.Inputs[32] := 0; END_IF;
   IF "IN_3-0.3" THEN "MODBUS".PLC_ports.Inputs[33] := 1; END_IF;
   IF NOT "IN_3-0.3" THEN "MODBUS".PLC_ports.Inputs[33] := 0; END_IF;
   IF "IN_3-0.4" THEN "MODBUS".PLC_ports.Inputs[34] := 1; END_IF;
   IF NOT "IN_3-0.4" THEN "MODBUS".PLC_ports.Inputs[34] := 0; END_IF;
   IF "IN_3-0.5" THEN "MODBUS".PLC_ports.Inputs[35] := 1; END_IF;
   IF NOT "IN_3-0.5" THEN "MODBUS".PLC_ports.Inputs[35] := 0; END_IF;
   IF "IN_3-0.6" THEN "MODBUS".PLC_ports.Inputs[36] := 1; END_IF;
   IF NOT "IN_3-0.6" THEN "MODBUS".PLC_ports.Inputs[36] := 0; END_IF;
   IF "IN_3-0.7" THEN "MODBUS".PLC_ports.Inputs[37] := 1; END_IF;
   IF NOT "IN_3-0.7" THEN "MODBUS".PLC_ports.Inputs[37] := 0; END_IF;
   IF "IN_3-1.0" THEN "MODBUS".PLC_ports.Inputs[38] := 1; END_IF;
   IF NOT "IN_3-1.0" THEN "MODBUS".PLC_ports.Inputs[38] := 0; END_IF;
   IF "IN_3-1.1" THEN "MODBUS".PLC_ports.Inputs[39] := 1; END_IF;
   IF NOT "IN_3-1.1" THEN "MODBUS".PLC_ports.Inputs[39] := 0; END_IF;
   IF "IN_3-1.2" THEN "MODBUS".PLC_ports.Inputs[40] := 1; END_IF;
   IF NOT "IN_3-1.2" THEN "MODBUS".PLC_ports.Inputs[40] := 0; END_IF;
   IF "IN_3-1.3" THEN "MODBUS".PLC_ports.Inputs[41] := 1; END_IF;
   IF NOT "IN_3-1.3" THEN "MODBUS".PLC_ports.Inputs[41] := 0; END_IF;
   IF "IN_3-1.4" THEN "MODBUS".PLC_ports.Inputs[42] := 1; END_IF;
   IF NOT "IN_3-1.4" THEN "MODBUS".PLC_ports.Inputs[42] := 0; END_IF;
   IF "IN_3-1.5" THEN "MODBUS".PLC_ports.Inputs[43] := 1; END_IF;
   IF NOT "IN_3-1.5" THEN "MODBUS".PLC_ports.Inputs[43] := 0; END_IF;
   IF "IN_3-1.6" THEN "MODBUS".PLC_ports.Inputs[44] := 1; END_IF;
   IF NOT "IN_3-1.6" THEN "MODBUS".PLC_ports.Inputs[44] := 0; END_IF;
   IF "IN_3-1.7" THEN "MODBUS".PLC_ports.Inputs[45] := 1; END_IF;
   IF NOT "IN_3-1.7" THEN "MODBUS".PLC_ports.Inputs[45] := 0; END_IF;
END_REGION

REGION Network 4
   // Входы 4 блока, Siemens SM-1223
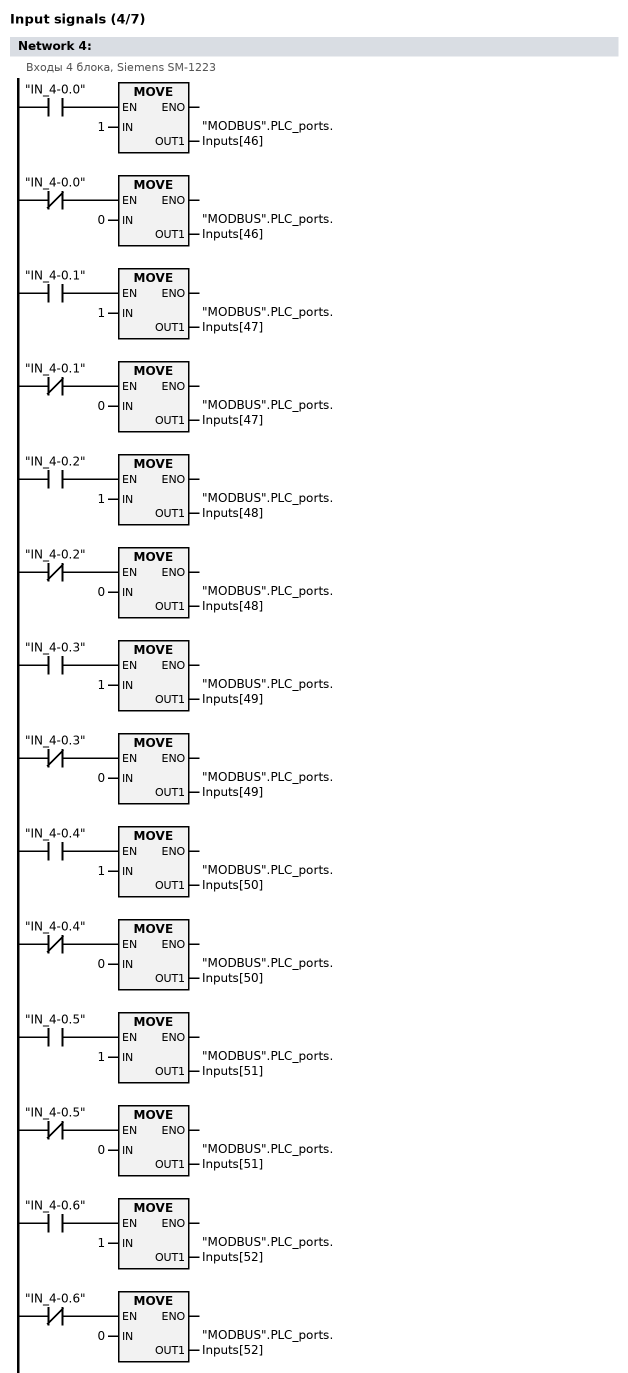
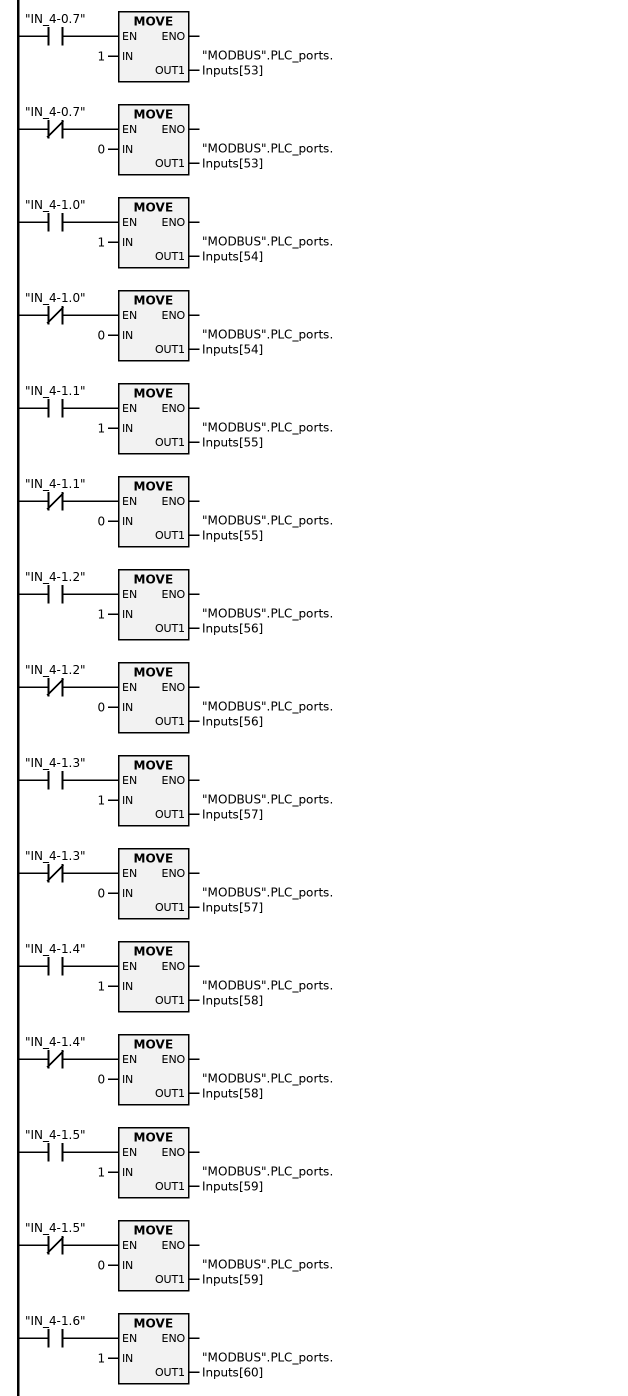
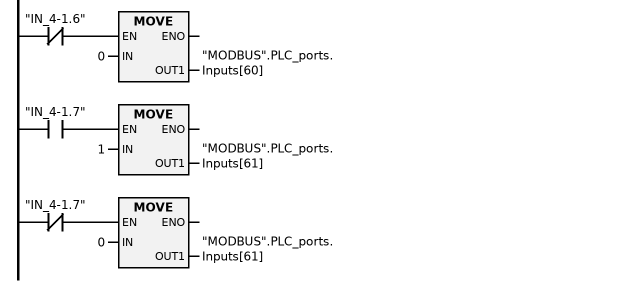
   RUNG wire#powerrail
      Contact( "IN_4-0.0" )
      Move(in := 1, out1 => "MODBUS".PLC_ports.Inputs[46])
   END_RUNG
   RUNG wire#powerrail
      I_Contact( "IN_4-0.0" )
      Move(in := 0, out1 => "MODBUS".PLC_ports.Inputs[46])
   END_RUNG
   RUNG wire#powerrail
      Contact( "IN_4-0.1" )
      Move(in := 1, out1 => "MODBUS".PLC_ports.Inputs[47])
   END_RUNG
   RUNG wire#powerrail
      I_Contact( "IN_4-0.1" )
      Move(in := 0, out1 => "MODBUS".PLC_ports.Inputs[47])
   END_RUNG
   RUNG wire#powerrail
      Contact( "IN_4-0.2" )
      Move(in := 1, out1 => "MODBUS".PLC_ports.Inputs[48])
   END_RUNG
   RUNG wire#powerrail
      I_Contact( "IN_4-0.2" )
      Move(in := 0, out1 => "MODBUS".PLC_ports.Inputs[48])
   END_RUNG
   RUNG wire#powerrail
      Contact( "IN_4-0.3" )
      Move(in := 1, out1 => "MODBUS".PLC_ports.Inputs[49])
   END_RUNG
   RUNG wire#powerrail
      I_Contact( "IN_4-0.3" )
      Move(in := 0, out1 => "MODBUS".PLC_ports.Inputs[49])
   END_RUNG
   RUNG wire#powerrail
      Contact( "IN_4-0.4" )
      Move(in := 1, out1 => "MODBUS".PLC_ports.Inputs[50])
   END_RUNG
   RUNG wire#powerrail
      I_Contact( "IN_4-0.4" )
      Move(in := 0, out1 => "MODBUS".PLC_ports.Inputs[50])
   END_RUNG
   RUNG wire#powerrail
      Contact( "IN_4-0.5" )
      Move(in := 1, out1 => "MODBUS".PLC_ports.Inputs[51])
   END_RUNG
   RUNG wire#powerrail
      I_Contact( "IN_4-0.5" )
      Move(in := 0, out1 => "MODBUS".PLC_ports.Inputs[51])
   END_RUNG
   RUNG wire#powerrail
      Contact( "IN_4-0.6" )
      Move(in := 1, out1 => "MODBUS".PLC_ports.Inputs[52])
   END_RUNG
   RUNG wire#powerrail
      I_Contact( "IN_4-0.6" )
      Move(in := 0, out1 => "MODBUS".PLC_ports.Inputs[52])
   END_RUNG
   RUNG wire#powerrail
      Contact( "IN_4-0.7" )
      Move(in := 1, out1 => "MODBUS".PLC_ports.Inputs[53])
   END_RUNG
   RUNG wire#powerrail
      I_Contact( "IN_4-0.7" )
      Move(in := 0, out1 => "MODBUS".PLC_ports.Inputs[53])
   END_RUNG
   RUNG wire#powerrail
      Contact( "IN_4-1.0" )
      Move(in := 1, out1 => "MODBUS".PLC_ports.Inputs[54])
   END_RUNG
   RUNG wire#powerrail
      I_Contact( "IN_4-1.0" )
      Move(in := 0, out1 => "MODBUS".PLC_ports.Inputs[54])
   END_RUNG
   RUNG wire#powerrail
      Contact( "IN_4-1.1" )
      Move(in := 1, out1 => "MODBUS".PLC_ports.Inputs[55])
   END_RUNG
   RUNG wire#powerrail
      I_Contact( "IN_4-1.1" )
      Move(in := 0, out1 => "MODBUS".PLC_ports.Inputs[55])
   END_RUNG
   RUNG wire#powerrail
      Contact( "IN_4-1.2" )
      Move(in := 1, out1 => "MODBUS".PLC_ports.Inputs[56])
   END_RUNG
   RUNG wire#powerrail
      I_Contact( "IN_4-1.2" )
      Move(in := 0, out1 => "MODBUS".PLC_ports.Inputs[56])
   END_RUNG
   RUNG wire#powerrail
      Contact( "IN_4-1.3" )
      Move(in := 1, out1 => "MODBUS".PLC_ports.Inputs[57])
   END_RUNG
   RUNG wire#powerrail
      I_Contact( "IN_4-1.3" )
      Move(in := 0, out1 => "MODBUS".PLC_ports.Inputs[57])
   END_RUNG
   RUNG wire#powerrail
      Contact( "IN_4-1.4" )
      Move(in := 1, out1 => "MODBUS".PLC_ports.Inputs[58])
   END_RUNG
   RUNG wire#powerrail
      I_Contact( "IN_4-1.4" )
      Move(in := 0, out1 => "MODBUS".PLC_ports.Inputs[58])
   END_RUNG
   RUNG wire#powerrail
      Contact( "IN_4-1.5" )
      Move(in := 1, out1 => "MODBUS".PLC_ports.Inputs[59])
   END_RUNG
   RUNG wire#powerrail
      I_Contact( "IN_4-1.5" )
      Move(in := 0, out1 => "MODBUS".PLC_ports.Inputs[59])
   END_RUNG
   RUNG wire#powerrail
      Contact( "IN_4-1.6" )
      Move(in := 1, out1 => "MODBUS".PLC_ports.Inputs[60])
   END_RUNG
   RUNG wire#powerrail
      I_Contact( "IN_4-1.6" )
      Move(in := 0, out1 => "MODBUS".PLC_ports.Inputs[60])
   END_RUNG
   RUNG wire#powerrail
      Contact( "IN_4-1.7" )
      Move(in := 1, out1 => "MODBUS".PLC_ports.Inputs[61])
   END_RUNG
   RUNG wire#powerrail
      I_Contact( "IN_4-1.7" )
      Move(in := 0, out1 => "MODBUS".PLC_ports.Inputs[61])
   END_RUNG
   // the same network as SCL:
   IF "IN_4-0.0" THEN "MODBUS".PLC_ports.Inputs[46] := 1; END_IF;
   IF NOT "IN_4-0.0" THEN "MODBUS".PLC_ports.Inputs[46] := 0; END_IF;
   IF "IN_4-0.1" THEN "MODBUS".PLC_ports.Inputs[47] := 1; END_IF;
   IF NOT "IN_4-0.1" THEN "MODBUS".PLC_ports.Inputs[47] := 0; END_IF;
   IF "IN_4-0.2" THEN "MODBUS".PLC_ports.Inputs[48] := 1; END_IF;
   IF NOT "IN_4-0.2" THEN "MODBUS".PLC_ports.Inputs[48] := 0; END_IF;
   IF "IN_4-0.3" THEN "MODBUS".PLC_ports.Inputs[49] := 1; END_IF;
   IF NOT "IN_4-0.3" THEN "MODBUS".PLC_ports.Inputs[49] := 0; END_IF;
   IF "IN_4-0.4" THEN "MODBUS".PLC_ports.Inputs[50] := 1; END_IF;
   IF NOT "IN_4-0.4" THEN "MODBUS".PLC_ports.Inputs[50] := 0; END_IF;
   IF "IN_4-0.5" THEN "MODBUS".PLC_ports.Inputs[51] := 1; END_IF;
   IF NOT "IN_4-0.5" THEN "MODBUS".PLC_ports.Inputs[51] := 0; END_IF;
   IF "IN_4-0.6" THEN "MODBUS".PLC_ports.Inputs[52] := 1; END_IF;
   IF NOT "IN_4-0.6" THEN "MODBUS".PLC_ports.Inputs[52] := 0; END_IF;
   IF "IN_4-0.7" THEN "MODBUS".PLC_ports.Inputs[53] := 1; END_IF;
   IF NOT "IN_4-0.7" THEN "MODBUS".PLC_ports.Inputs[53] := 0; END_IF;
   IF "IN_4-1.0" THEN "MODBUS".PLC_ports.Inputs[54] := 1; END_IF;
   IF NOT "IN_4-1.0" THEN "MODBUS".PLC_ports.Inputs[54] := 0; END_IF;
   IF "IN_4-1.1" THEN "MODBUS".PLC_ports.Inputs[55] := 1; END_IF;
   IF NOT "IN_4-1.1" THEN "MODBUS".PLC_ports.Inputs[55] := 0; END_IF;
   IF "IN_4-1.2" THEN "MODBUS".PLC_ports.Inputs[56] := 1; END_IF;
   IF NOT "IN_4-1.2" THEN "MODBUS".PLC_ports.Inputs[56] := 0; END_IF;
   IF "IN_4-1.3" THEN "MODBUS".PLC_ports.Inputs[57] := 1; END_IF;
   IF NOT "IN_4-1.3" THEN "MODBUS".PLC_ports.Inputs[57] := 0; END_IF;
   IF "IN_4-1.4" THEN "MODBUS".PLC_ports.Inputs[58] := 1; END_IF;
   IF NOT "IN_4-1.4" THEN "MODBUS".PLC_ports.Inputs[58] := 0; END_IF;
   IF "IN_4-1.5" THEN "MODBUS".PLC_ports.Inputs[59] := 1; END_IF;
   IF NOT "IN_4-1.5" THEN "MODBUS".PLC_ports.Inputs[59] := 0; END_IF;
   IF "IN_4-1.6" THEN "MODBUS".PLC_ports.Inputs[60] := 1; END_IF;
   IF NOT "IN_4-1.6" THEN "MODBUS".PLC_ports.Inputs[60] := 0; END_IF;
   IF "IN_4-1.7" THEN "MODBUS".PLC_ports.Inputs[61] := 1; END_IF;
   IF NOT "IN_4-1.7" THEN "MODBUS".PLC_ports.Inputs[61] := 0; END_IF;
END_REGION

REGION Network 5
   // Входы 5 блока, Siemens SM-1223
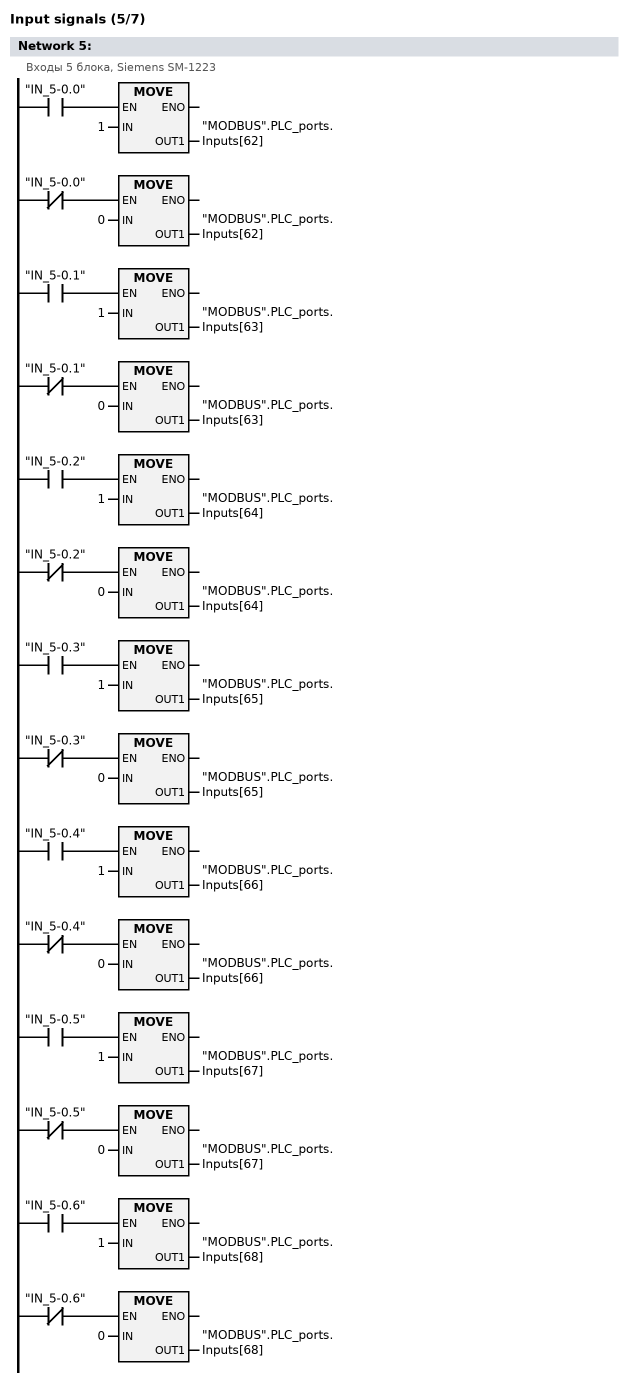
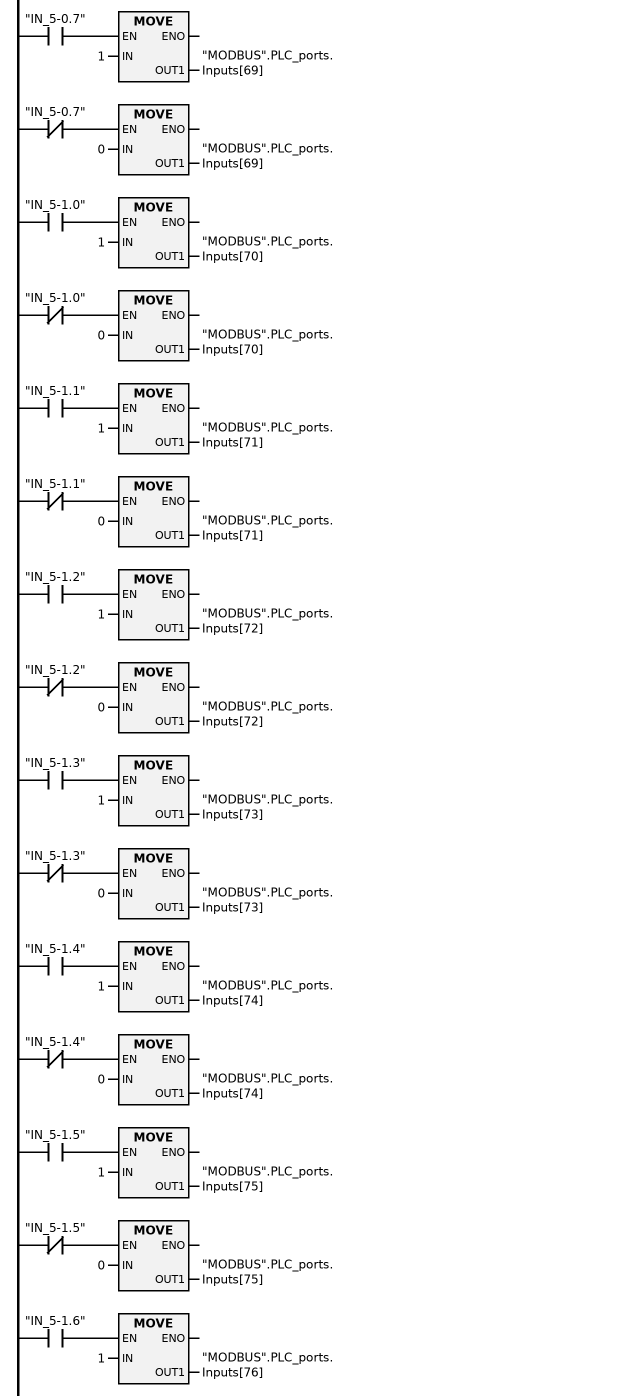
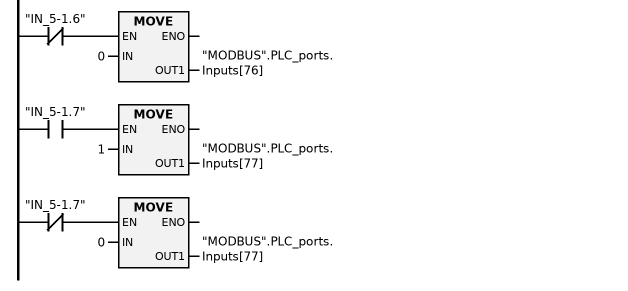
   RUNG wire#powerrail
      Contact( "IN_5-0.0" )
      Move(in := 1, out1 => "MODBUS".PLC_ports.Inputs[62])
   END_RUNG
   RUNG wire#powerrail
      I_Contact( "IN_5-0.0" )
      Move(in := 0, out1 => "MODBUS".PLC_ports.Inputs[62])
   END_RUNG
   RUNG wire#powerrail
      Contact( "IN_5-0.1" )
      Move(in := 1, out1 => "MODBUS".PLC_ports.Inputs[63])
   END_RUNG
   RUNG wire#powerrail
      I_Contact( "IN_5-0.1" )
      Move(in := 0, out1 => "MODBUS".PLC_ports.Inputs[63])
   END_RUNG
   RUNG wire#powerrail
      Contact( "IN_5-0.2" )
      Move(in := 1, out1 => "MODBUS".PLC_ports.Inputs[64])
   END_RUNG
   RUNG wire#powerrail
      I_Contact( "IN_5-0.2" )
      Move(in := 0, out1 => "MODBUS".PLC_ports.Inputs[64])
   END_RUNG
   RUNG wire#powerrail
      Contact( "IN_5-0.3" )
      Move(in := 1, out1 => "MODBUS".PLC_ports.Inputs[65])
   END_RUNG
   RUNG wire#powerrail
      I_Contact( "IN_5-0.3" )
      Move(in := 0, out1 => "MODBUS".PLC_ports.Inputs[65])
   END_RUNG
   RUNG wire#powerrail
      Contact( "IN_5-0.4" )
      Move(in := 1, out1 => "MODBUS".PLC_ports.Inputs[66])
   END_RUNG
   RUNG wire#powerrail
      I_Contact( "IN_5-0.4" )
      Move(in := 0, out1 => "MODBUS".PLC_ports.Inputs[66])
   END_RUNG
   RUNG wire#powerrail
      Contact( "IN_5-0.5" )
      Move(in := 1, out1 => "MODBUS".PLC_ports.Inputs[67])
   END_RUNG
   RUNG wire#powerrail
      I_Contact( "IN_5-0.5" )
      Move(in := 0, out1 => "MODBUS".PLC_ports.Inputs[67])
   END_RUNG
   RUNG wire#powerrail
      Contact( "IN_5-0.6" )
      Move(in := 1, out1 => "MODBUS".PLC_ports.Inputs[68])
   END_RUNG
   RUNG wire#powerrail
      I_Contact( "IN_5-0.6" )
      Move(in := 0, out1 => "MODBUS".PLC_ports.Inputs[68])
   END_RUNG
   RUNG wire#powerrail
      Contact( "IN_5-0.7" )
      Move(in := 1, out1 => "MODBUS".PLC_ports.Inputs[69])
   END_RUNG
   RUNG wire#powerrail
      I_Contact( "IN_5-0.7" )
      Move(in := 0, out1 => "MODBUS".PLC_ports.Inputs[69])
   END_RUNG
   RUNG wire#powerrail
      Contact( "IN_5-1.0" )
      Move(in := 1, out1 => "MODBUS".PLC_ports.Inputs[70])
   END_RUNG
   RUNG wire#powerrail
      I_Contact( "IN_5-1.0" )
      Move(in := 0, out1 => "MODBUS".PLC_ports.Inputs[70])
   END_RUNG
   RUNG wire#powerrail
      Contact( "IN_5-1.1" )
      Move(in := 1, out1 => "MODBUS".PLC_ports.Inputs[71])
   END_RUNG
   RUNG wire#powerrail
      I_Contact( "IN_5-1.1" )
      Move(in := 0, out1 => "MODBUS".PLC_ports.Inputs[71])
   END_RUNG
   RUNG wire#powerrail
      Contact( "IN_5-1.2" )
      Move(in := 1, out1 => "MODBUS".PLC_ports.Inputs[72])
   END_RUNG
   RUNG wire#powerrail
      I_Contact( "IN_5-1.2" )
      Move(in := 0, out1 => "MODBUS".PLC_ports.Inputs[72])
   END_RUNG
   RUNG wire#powerrail
      Contact( "IN_5-1.3" )
      Move(in := 1, out1 => "MODBUS".PLC_ports.Inputs[73])
   END_RUNG
   RUNG wire#powerrail
      I_Contact( "IN_5-1.3" )
      Move(in := 0, out1 => "MODBUS".PLC_ports.Inputs[73])
   END_RUNG
   RUNG wire#powerrail
      Contact( "IN_5-1.4" )
      Move(in := 1, out1 => "MODBUS".PLC_ports.Inputs[74])
   END_RUNG
   RUNG wire#powerrail
      I_Contact( "IN_5-1.4" )
      Move(in := 0, out1 => "MODBUS".PLC_ports.Inputs[74])
   END_RUNG
   RUNG wire#powerrail
      Contact( "IN_5-1.5" )
      Move(in := 1, out1 => "MODBUS".PLC_ports.Inputs[75])
   END_RUNG
   RUNG wire#powerrail
      I_Contact( "IN_5-1.5" )
      Move(in := 0, out1 => "MODBUS".PLC_ports.Inputs[75])
   END_RUNG
   RUNG wire#powerrail
      Contact( "IN_5-1.6" )
      Move(in := 1, out1 => "MODBUS".PLC_ports.Inputs[76])
   END_RUNG
   RUNG wire#powerrail
      I_Contact( "IN_5-1.6" )
      Move(in := 0, out1 => "MODBUS".PLC_ports.Inputs[76])
   END_RUNG
   RUNG wire#powerrail
      Contact( "IN_5-1.7" )
      Move(in := 1, out1 => "MODBUS".PLC_ports.Inputs[77])
   END_RUNG
   RUNG wire#powerrail
      I_Contact( "IN_5-1.7" )
      Move(in := 0, out1 => "MODBUS".PLC_ports.Inputs[77])
   END_RUNG
   // the same network as SCL:
   IF "IN_5-0.0" THEN "MODBUS".PLC_ports.Inputs[62] := 1; END_IF;
   IF NOT "IN_5-0.0" THEN "MODBUS".PLC_ports.Inputs[62] := 0; END_IF;
   IF "IN_5-0.1" THEN "MODBUS".PLC_ports.Inputs[63] := 1; END_IF;
   IF NOT "IN_5-0.1" THEN "MODBUS".PLC_ports.Inputs[63] := 0; END_IF;
   IF "IN_5-0.2" THEN "MODBUS".PLC_ports.Inputs[64] := 1; END_IF;
   IF NOT "IN_5-0.2" THEN "MODBUS".PLC_ports.Inputs[64] := 0; END_IF;
   IF "IN_5-0.3" THEN "MODBUS".PLC_ports.Inputs[65] := 1; END_IF;
   IF NOT "IN_5-0.3" THEN "MODBUS".PLC_ports.Inputs[65] := 0; END_IF;
   IF "IN_5-0.4" THEN "MODBUS".PLC_ports.Inputs[66] := 1; END_IF;
   IF NOT "IN_5-0.4" THEN "MODBUS".PLC_ports.Inputs[66] := 0; END_IF;
   IF "IN_5-0.5" THEN "MODBUS".PLC_ports.Inputs[67] := 1; END_IF;
   IF NOT "IN_5-0.5" THEN "MODBUS".PLC_ports.Inputs[67] := 0; END_IF;
   IF "IN_5-0.6" THEN "MODBUS".PLC_ports.Inputs[68] := 1; END_IF;
   IF NOT "IN_5-0.6" THEN "MODBUS".PLC_ports.Inputs[68] := 0; END_IF;
   IF "IN_5-0.7" THEN "MODBUS".PLC_ports.Inputs[69] := 1; END_IF;
   IF NOT "IN_5-0.7" THEN "MODBUS".PLC_ports.Inputs[69] := 0; END_IF;
   IF "IN_5-1.0" THEN "MODBUS".PLC_ports.Inputs[70] := 1; END_IF;
   IF NOT "IN_5-1.0" THEN "MODBUS".PLC_ports.Inputs[70] := 0; END_IF;
   IF "IN_5-1.1" THEN "MODBUS".PLC_ports.Inputs[71] := 1; END_IF;
   IF NOT "IN_5-1.1" THEN "MODBUS".PLC_ports.Inputs[71] := 0; END_IF;
   IF "IN_5-1.2" THEN "MODBUS".PLC_ports.Inputs[72] := 1; END_IF;
   IF NOT "IN_5-1.2" THEN "MODBUS".PLC_ports.Inputs[72] := 0; END_IF;
   IF "IN_5-1.3" THEN "MODBUS".PLC_ports.Inputs[73] := 1; END_IF;
   IF NOT "IN_5-1.3" THEN "MODBUS".PLC_ports.Inputs[73] := 0; END_IF;
   IF "IN_5-1.4" THEN "MODBUS".PLC_ports.Inputs[74] := 1; END_IF;
   IF NOT "IN_5-1.4" THEN "MODBUS".PLC_ports.Inputs[74] := 0; END_IF;
   IF "IN_5-1.5" THEN "MODBUS".PLC_ports.Inputs[75] := 1; END_IF;
   IF NOT "IN_5-1.5" THEN "MODBUS".PLC_ports.Inputs[75] := 0; END_IF;
   IF "IN_5-1.6" THEN "MODBUS".PLC_ports.Inputs[76] := 1; END_IF;
   IF NOT "IN_5-1.6" THEN "MODBUS".PLC_ports.Inputs[76] := 0; END_IF;
   IF "IN_5-1.7" THEN "MODBUS".PLC_ports.Inputs[77] := 1; END_IF;
   IF NOT "IN_5-1.7" THEN "MODBUS".PLC_ports.Inputs[77] := 0; END_IF;
END_REGION

REGION Network 6
   // Входы 6 блока, Siemens SM-1223
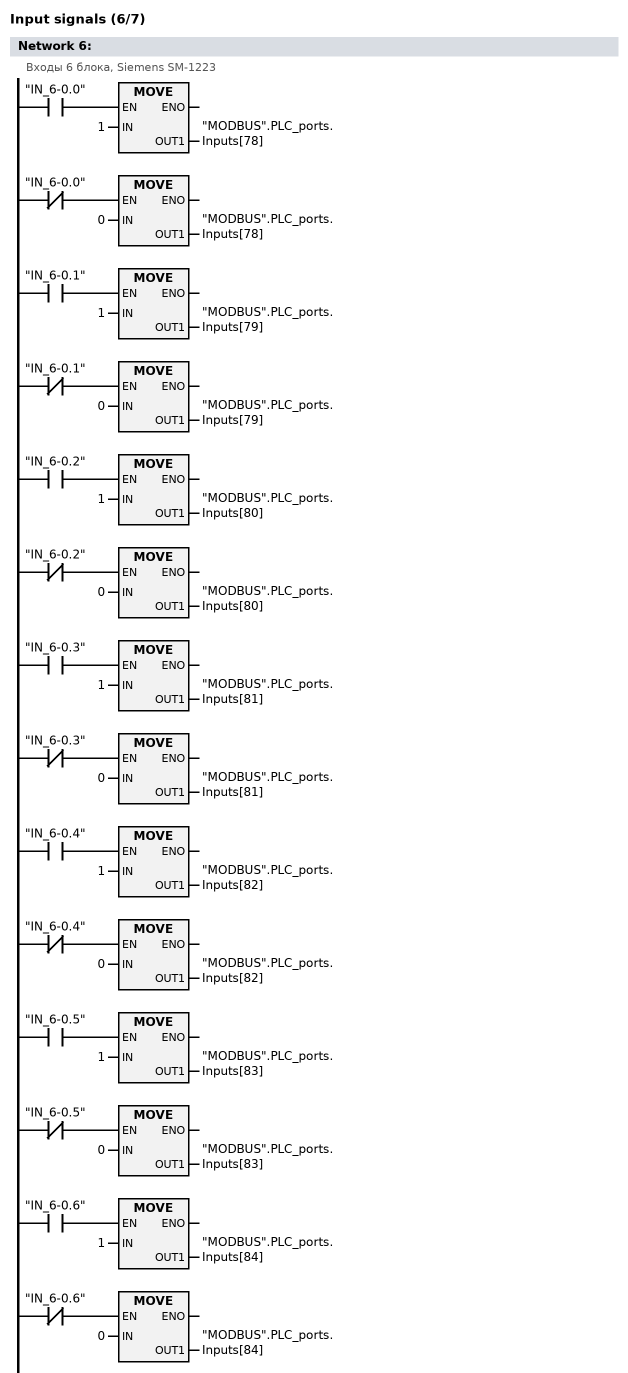
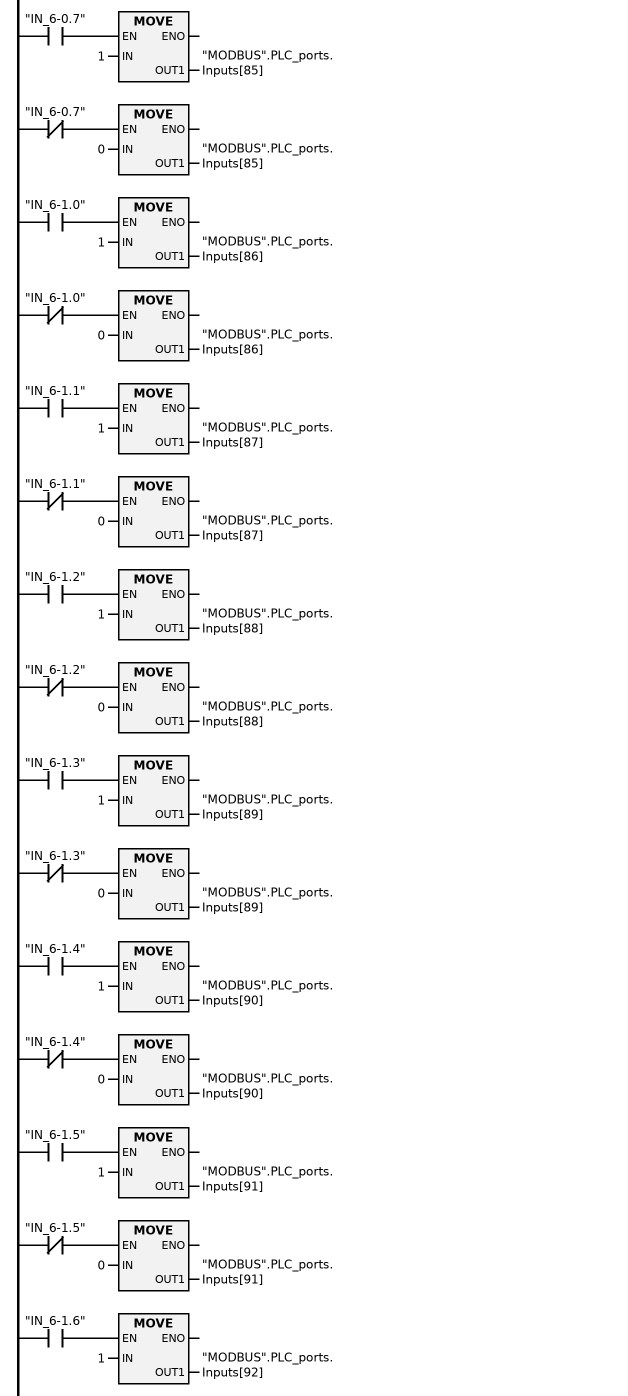
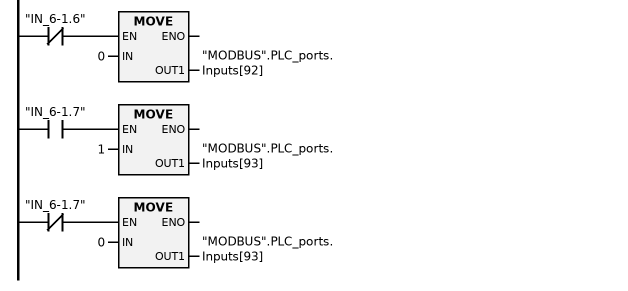
   RUNG wire#powerrail
      Contact( "IN_6-0.0" )
      Move(in := 1, out1 => "MODBUS".PLC_ports.Inputs[78])
   END_RUNG
   RUNG wire#powerrail
      I_Contact( "IN_6-0.0" )
      Move(in := 0, out1 => "MODBUS".PLC_ports.Inputs[78])
   END_RUNG
   RUNG wire#powerrail
      Contact( "IN_6-0.1" )
      Move(in := 1, out1 => "MODBUS".PLC_ports.Inputs[79])
   END_RUNG
   RUNG wire#powerrail
      I_Contact( "IN_6-0.1" )
      Move(in := 0, out1 => "MODBUS".PLC_ports.Inputs[79])
   END_RUNG
   RUNG wire#powerrail
      Contact( "IN_6-0.2" )
      Move(in := 1, out1 => "MODBUS".PLC_ports.Inputs[80])
   END_RUNG
   RUNG wire#powerrail
      I_Contact( "IN_6-0.2" )
      Move(in := 0, out1 => "MODBUS".PLC_ports.Inputs[80])
   END_RUNG
   RUNG wire#powerrail
      Contact( "IN_6-0.3" )
      Move(in := 1, out1 => "MODBUS".PLC_ports.Inputs[81])
   END_RUNG
   RUNG wire#powerrail
      I_Contact( "IN_6-0.3" )
      Move(in := 0, out1 => "MODBUS".PLC_ports.Inputs[81])
   END_RUNG
   RUNG wire#powerrail
      Contact( "IN_6-0.4" )
      Move(in := 1, out1 => "MODBUS".PLC_ports.Inputs[82])
   END_RUNG
   RUNG wire#powerrail
      I_Contact( "IN_6-0.4" )
      Move(in := 0, out1 => "MODBUS".PLC_ports.Inputs[82])
   END_RUNG
   RUNG wire#powerrail
      Contact( "IN_6-0.5" )
      Move(in := 1, out1 => "MODBUS".PLC_ports.Inputs[83])
   END_RUNG
   RUNG wire#powerrail
      I_Contact( "IN_6-0.5" )
      Move(in := 0, out1 => "MODBUS".PLC_ports.Inputs[83])
   END_RUNG
   RUNG wire#powerrail
      Contact( "IN_6-0.6" )
      Move(in := 1, out1 => "MODBUS".PLC_ports.Inputs[84])
   END_RUNG
   RUNG wire#powerrail
      I_Contact( "IN_6-0.6" )
      Move(in := 0, out1 => "MODBUS".PLC_ports.Inputs[84])
   END_RUNG
   RUNG wire#powerrail
      Contact( "IN_6-0.7" )
      Move(in := 1, out1 => "MODBUS".PLC_ports.Inputs[85])
   END_RUNG
   RUNG wire#powerrail
      I_Contact( "IN_6-0.7" )
      Move(in := 0, out1 => "MODBUS".PLC_ports.Inputs[85])
   END_RUNG
   RUNG wire#powerrail
      Contact( "IN_6-1.0" )
      Move(in := 1, out1 => "MODBUS".PLC_ports.Inputs[86])
   END_RUNG
   RUNG wire#powerrail
      I_Contact( "IN_6-1.0" )
      Move(in := 0, out1 => "MODBUS".PLC_ports.Inputs[86])
   END_RUNG
   RUNG wire#powerrail
      Contact( "IN_6-1.1" )
      Move(in := 1, out1 => "MODBUS".PLC_ports.Inputs[87])
   END_RUNG
   RUNG wire#powerrail
      I_Contact( "IN_6-1.1" )
      Move(in := 0, out1 => "MODBUS".PLC_ports.Inputs[87])
   END_RUNG
   RUNG wire#powerrail
      Contact( "IN_6-1.2" )
      Move(in := 1, out1 => "MODBUS".PLC_ports.Inputs[88])
   END_RUNG
   RUNG wire#powerrail
      I_Contact( "IN_6-1.2" )
      Move(in := 0, out1 => "MODBUS".PLC_ports.Inputs[88])
   END_RUNG
   RUNG wire#powerrail
      Contact( "IN_6-1.3" )
      Move(in := 1, out1 => "MODBUS".PLC_ports.Inputs[89])
   END_RUNG
   RUNG wire#powerrail
      I_Contact( "IN_6-1.3" )
      Move(in := 0, out1 => "MODBUS".PLC_ports.Inputs[89])
   END_RUNG
   RUNG wire#powerrail
      Contact( "IN_6-1.4" )
      Move(in := 1, out1 => "MODBUS".PLC_ports.Inputs[90])
   END_RUNG
   RUNG wire#powerrail
      I_Contact( "IN_6-1.4" )
      Move(in := 0, out1 => "MODBUS".PLC_ports.Inputs[90])
   END_RUNG
   RUNG wire#powerrail
      Contact( "IN_6-1.5" )
      Move(in := 1, out1 => "MODBUS".PLC_ports.Inputs[91])
   END_RUNG
   RUNG wire#powerrail
      I_Contact( "IN_6-1.5" )
      Move(in := 0, out1 => "MODBUS".PLC_ports.Inputs[91])
   END_RUNG
   RUNG wire#powerrail
      Contact( "IN_6-1.6" )
      Move(in := 1, out1 => "MODBUS".PLC_ports.Inputs[92])
   END_RUNG
   RUNG wire#powerrail
      I_Contact( "IN_6-1.6" )
      Move(in := 0, out1 => "MODBUS".PLC_ports.Inputs[92])
   END_RUNG
   RUNG wire#powerrail
      Contact( "IN_6-1.7" )
      Move(in := 1, out1 => "MODBUS".PLC_ports.Inputs[93])
   END_RUNG
   RUNG wire#powerrail
      I_Contact( "IN_6-1.7" )
      Move(in := 0, out1 => "MODBUS".PLC_ports.Inputs[93])
   END_RUNG
   // the same network as SCL:
   IF "IN_6-0.0" THEN "MODBUS".PLC_ports.Inputs[78] := 1; END_IF;
   IF NOT "IN_6-0.0" THEN "MODBUS".PLC_ports.Inputs[78] := 0; END_IF;
   IF "IN_6-0.1" THEN "MODBUS".PLC_ports.Inputs[79] := 1; END_IF;
   IF NOT "IN_6-0.1" THEN "MODBUS".PLC_ports.Inputs[79] := 0; END_IF;
   IF "IN_6-0.2" THEN "MODBUS".PLC_ports.Inputs[80] := 1; END_IF;
   IF NOT "IN_6-0.2" THEN "MODBUS".PLC_ports.Inputs[80] := 0; END_IF;
   IF "IN_6-0.3" THEN "MODBUS".PLC_ports.Inputs[81] := 1; END_IF;
   IF NOT "IN_6-0.3" THEN "MODBUS".PLC_ports.Inputs[81] := 0; END_IF;
   IF "IN_6-0.4" THEN "MODBUS".PLC_ports.Inputs[82] := 1; END_IF;
   IF NOT "IN_6-0.4" THEN "MODBUS".PLC_ports.Inputs[82] := 0; END_IF;
   IF "IN_6-0.5" THEN "MODBUS".PLC_ports.Inputs[83] := 1; END_IF;
   IF NOT "IN_6-0.5" THEN "MODBUS".PLC_ports.Inputs[83] := 0; END_IF;
   IF "IN_6-0.6" THEN "MODBUS".PLC_ports.Inputs[84] := 1; END_IF;
   IF NOT "IN_6-0.6" THEN "MODBUS".PLC_ports.Inputs[84] := 0; END_IF;
   IF "IN_6-0.7" THEN "MODBUS".PLC_ports.Inputs[85] := 1; END_IF;
   IF NOT "IN_6-0.7" THEN "MODBUS".PLC_ports.Inputs[85] := 0; END_IF;
   IF "IN_6-1.0" THEN "MODBUS".PLC_ports.Inputs[86] := 1; END_IF;
   IF NOT "IN_6-1.0" THEN "MODBUS".PLC_ports.Inputs[86] := 0; END_IF;
   IF "IN_6-1.1" THEN "MODBUS".PLC_ports.Inputs[87] := 1; END_IF;
   IF NOT "IN_6-1.1" THEN "MODBUS".PLC_ports.Inputs[87] := 0; END_IF;
   IF "IN_6-1.2" THEN "MODBUS".PLC_ports.Inputs[88] := 1; END_IF;
   IF NOT "IN_6-1.2" THEN "MODBUS".PLC_ports.Inputs[88] := 0; END_IF;
   IF "IN_6-1.3" THEN "MODBUS".PLC_ports.Inputs[89] := 1; END_IF;
   IF NOT "IN_6-1.3" THEN "MODBUS".PLC_ports.Inputs[89] := 0; END_IF;
   IF "IN_6-1.4" THEN "MODBUS".PLC_ports.Inputs[90] := 1; END_IF;
   IF NOT "IN_6-1.4" THEN "MODBUS".PLC_ports.Inputs[90] := 0; END_IF;
   IF "IN_6-1.5" THEN "MODBUS".PLC_ports.Inputs[91] := 1; END_IF;
   IF NOT "IN_6-1.5" THEN "MODBUS".PLC_ports.Inputs[91] := 0; END_IF;
   IF "IN_6-1.6" THEN "MODBUS".PLC_ports.Inputs[92] := 1; END_IF;
   IF NOT "IN_6-1.6" THEN "MODBUS".PLC_ports.Inputs[92] := 0; END_IF;
   IF "IN_6-1.7" THEN "MODBUS".PLC_ports.Inputs[93] := 1; END_IF;
   IF NOT "IN_6-1.7" THEN "MODBUS".PLC_ports.Inputs[93] := 0; END_IF;
END_REGION

REGION Network 7
   // Входы 7 блока, Siemens SM-1223
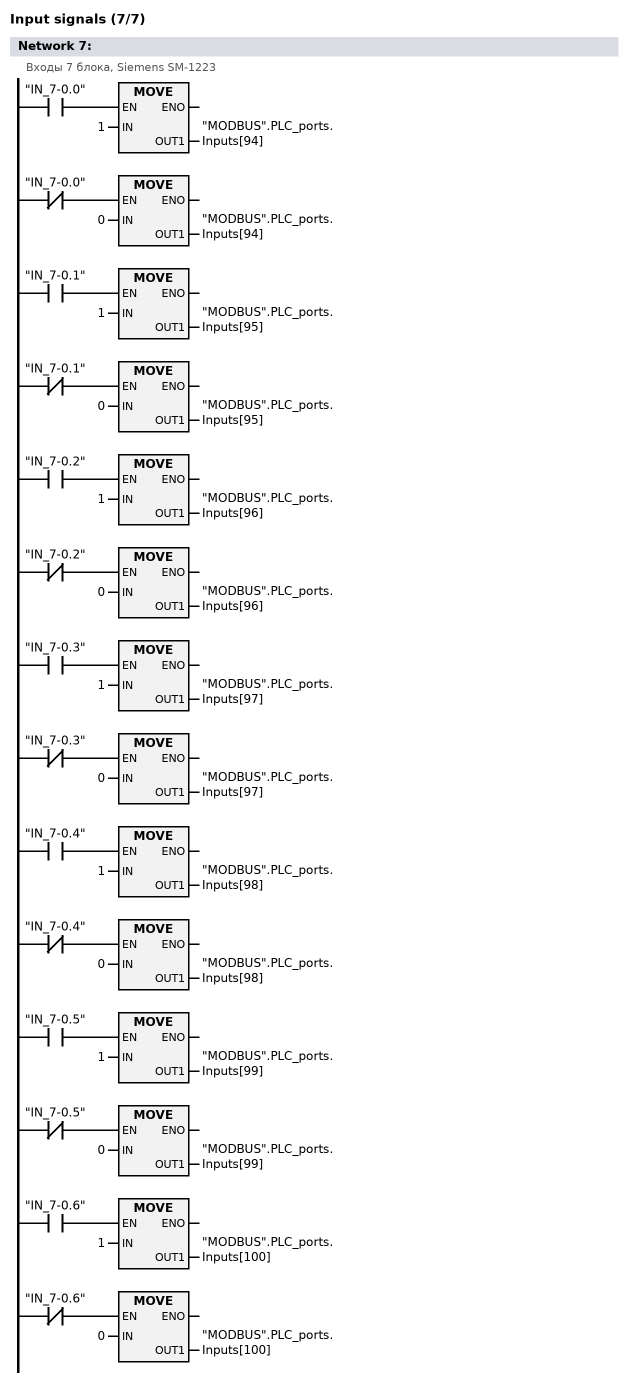
